// TwinCAT 3 PLC project Runtime
// ProgramVersion: 3.1.4026.14
// libraries:
//   Tc2_ControllerToolbox, * (Beckhoff Automation GmbH)
//   Tc2_ModbusSrv, * (Beckhoff Automation GmbH)
//   Tc2_Standard, * (Beckhoff Automation GmbH)
//   Tc2_System, * (Beckhoff Automation GmbH)
//   Tc2_Utilities, * (Beckhoff Automation GmbH)
//   Tc3_IotBase, * (Beckhoff Automation GmbH)
//   Tc3_Module, * (Beckhoff Automation GmbH)
// project tree:
//   DUTs/Algorithms/ stBESS.TcDUT, stCMD_SET.TcDUT, stCONV_UNION.TcDUT, stGRID_POS.TcDUT, stINVERTER.TcDUT, stMETER.TcDUT, stPF_POINT.TcDUT, stPOWER_PLANT.TcDUT, stPPC.TcDUT, stQV_POINT.TcDUT, stRECORD.TcDUT, stTIMESLOT.TcDUT
//   / FreqReg.TcTTO, PlcTask.TcTTO
//   GVLs/Algorithms/ GVL.TcGVL, GVL_Act_Pwr.TcGVL, GVL_Freq.TcGVL, GVL_Load_Following.TcGVL, GVL_Modules.TcGVL, GVL_React_Pwr.TcGVL, GVL_Voltage.TcGVL
//   POUs/ MAIN.TcPOU
//   POUs/Programs/Algorithms/Active power regulation/ Active_Power_Regulation.TcPOU, deltaActivePwr_Frequency_Regulation.TcPOU, FB_Frequency_Regulation.TcPOU, FB_Reach_SP_ActP.TcPOU
//   POUs/Programs/Algorithms/Automatic controls/ FF_BLOCK.TcPOU, Low_Pass_Filter.TcPOU, FB_PI_Setpoint.TcPOU
//   POUs/Programs/Algorithms/Cosmo Eco/ Calculate_Opt_SOC_Based_On_Conditions.TcPOU, Calculate_Opt_SOC_No_Decrease.TcPOU, Calculate_Set_Point_Normal_Conditions.TcPOU, No_Decrease.TcPOU, No_Increase.TcPOU, No_Limit.TcPOU, Pre_Lim.TcPOU, Static.TcPOU
//   POUs/Programs/Algorithms/Load Following/ FB_Load_Following.TcPOU
//   POUs/Programs/Algorithms/ FB_Load_From_DB.TcPOU, Main_Algorithm.TcPOU, FB_Module_Executor.TcPOU, outputQV_regulation.TcPOU, power_at_nominal_freq.TcPOU, Primary_Regulations.TcPOU, reactp_sp_from_pf.TcPOU, setpoint_acquired.TcPOU, sp_input_reducer.TcPOU
//   POUs/Programs/Algorithms/Meter/ Update_Virtual_Meter.TcPOU
//   POUs/Programs/Algorithms/Reactive power regulation/ deltaReactivePwr_Voltage_Regulation.TcPOU, FB_Hysteresis.TcPOU, FB_Map_QV.TcPOU, FB_Reach_SP_ReactP.TcPOU, FB_ReactivePwr_Voltage_Ctrl.TcPOU, Reactive_Power_Regulation.TcPOU
//   POUs/Programs/Engine/Inverter Comm/ Apply_Setpoint.TcPOU, FB_Check_Inverter_Health.TcPOU, FB_Command_Dispatcher.TcPOU, FB_Comm_Setup.TcPOU
//   POUs/Programs/Engine/ MQTT_TSO_Comm.TcPOU, FB_Read_Meter.TcPOU, FB_Setup_Meter_Comm.TcPOU

CONFIGURATION Runtime
    RESOURCE PLC ON TwinCAT3
        TASK FreqReg(INTERVAL := T#100000us, PRIORITY := 1);
        TASK PlcTask(INTERVAL := T#10ms, PRIORITY := 20);
        PROGRAM Primary_Regulations WITH FreqReg : Primary_Regulations;
        PROGRAM MAIN WITH PlcTask : MAIN;
    END_RESOURCE
END_CONFIGURATION

// ---- DUTs/Algorithms/stBESS.TcDUT
TYPE stBESS :
STRUCT
	
	soc: REAL; // [0, 1]
	capacity: REAL;
	available_power: REAL;
	
	max_tolerable_soc: REAL;
	min_tolerable_soc: REAL;
	
	soc_to_remove_sp: REAL;
	
	max_opt_soc: REAL;
	min_opt_soc: REAL;
	
	min_soc: REAL;
	efficiency: REAL;
	
	min_working_soc: REAL;
	
END_STRUCT
END_TYPE

// ---- DUTs/Algorithms/stCMD_SET.TcDUT
TYPE stCMD_SET :
STRUCT
	command_for_battery: REAL;
	plant_sp: REAL;
END_STRUCT
END_TYPE

// ---- DUTs/Algorithms/stCONV_UNION.TcDUT
TYPE stCONV_UNION :
UNION
	prod_real: REAL;
	prod_w: ARRAY[1..2] of WORD;
END_UNION
END_TYPE

// ---- DUTs/Algorithms/stGRID_POS.TcDUT
{attribute 'qualified_only'}
{attribute 'strict'}
TYPE stGRID_POS :
(
	poi := 0,
	pu := 1
);
END_TYPE

// ---- DUTs/Algorithms/stINVERTER.TcDUT
TYPE stINVERTER :
STRUCT
	/// INVERTER STATUS
	health: UINT;	// 1 = health, 0 = fault
	
	/// ACTIVE POWER ///
	current_sp: REAL;
	target_prod: REAL; 
	active_pwr_nominal_pwr: REAL;
	sp_mem: REAL;
	sp_mem_q: REAL;
	
	/// REACTIVE POWER /// 
	current_sp_q: REAL;
	reactive_pwr_nominal_pwr: REAL;
	
	/// MODBUS COMM
	tcp_port: UINT;
	unit_id: BYTE;
	server_ip_addr: STRING(255);
	n_quantity_act_pwr: WORD;
	mb_addr_act_pwr: WORD;
	n_quantity_react_pwr: WORD;
	mb_addr_react_pwr: WORD;
	mb_h_addr: WORD;
	health_quantity: WORD;
	
	read_done: BOOL := FALSE;
	read_state: UINT := 0;
	
	write_done: BOOL := TRUE;
	write_state: UINT := 0;
	
	wBusy_actp: BOOL;
	wBusy_reactp: BOOL;
	
	comm_state: UINT;
	
END_STRUCT
END_TYPE

// ---- DUTs/Algorithms/stMETER.TcDUT
TYPE stMETER :
STRUCT
	
	/// MODBUS ///
	tcp_port: UINT := 9501;
	unit_id: BYTE;
	server_ip_addr: STRING(255);
	
	/// ACTIVE POWER ///
	frequency: REAL;
	active_power_prod: REAL;
	active_power_sp: REAL;
	nQuantity_Act_Pwr: WORD;
	nMBAddr_Act_Pwr: WORD;
	
	/// REACTIVE POWER ///
	reactive_power_prod: REAL;
	reactive_power_sp: REAL;
	measured_voltage: REAL;
	nQuantity_React_Pwr: WORD;
	nMBAddr_React_Pwr: WORD;
	
	pos: stGRID_POS;	// questa variabile specifica dove è installato l'inverter e consente di distinguere meter di griglia (poi) da meter d'impianto (pu)
	
END_STRUCT
END_TYPE

// ---- DUTs/Algorithms/stPF_POINT.TcDUT
TYPE stPF_POINT :
STRUCT
	active_power: REAL;
	frequency: REAL;
END_STRUCT
END_TYPE

// ---- DUTs/Algorithms/stPOWER_PLANT.TcDUT
TYPE stPOWER_PLANT :
STRUCT
	// TO DO: in futuro, spostare tutte le variabili riguardanti l'impianto qui dentro
	safety_margin: REAL;
	max_power_increase: REAL; 
	ramp_limit: REAL; //[kW/min]
	sample_time: REAL;
	current_time: REAL;
	
	max_kw_change_3s: REAL;		// TO DO: questa variabile è rappresenta un'ulteriore limitazione che può essere presente in alcuni casi
	
	nominal_power: REAL := 1E4;
	
	avg_prod: REAL; 	// floating average level of production
	avg_prod_diff: REAL;
	
	avg_prod_3h: REAL; 	// average level of production over 3 hours. This variable is specific for the CosmoEco project 
	std_deviation_prod: REAL;
	
END_STRUCT
END_TYPE

// ---- DUTs/Algorithms/stPPC.TcDUT
TYPE stPPC :
STRUCT
	
	START: BOOL := TRUE;	
	MANUAL_MODE: BOOL;  /// FIELD OPERATOR ///
	AUTO_MODE: BOOL;	/// CONTROL ROOM ///
	REMOTE_MODE: BOOL := TRUE;	/// TSO via MQTT///
	
	actp_freq_reg_enabled: BOOL := FALSE;
	active_power_ctrl_enabled: BOOL := TRUE;
	reactive_power_ctrl_enabled: BOOL := TRUE;
	qv_ctrl_enabled: BOOL := TRUE;
	power_factor_ctrl_enabled: BOOL := FALSE;
	load_following_enabled: BOOL := FALSE;
	
	timeslot: stTIMESLOT;
	
END_STRUCT
END_TYPE

// ---- DUTs/Algorithms/stQV_POINT.TcDUT
TYPE stQV_POINT :
STRUCT
	voltage_ratio: REAL;
	q_pnd_ratio: REAL;
END_STRUCT
END_TYPE

// ---- DUTs/Algorithms/stRECORD.TcDUT
TYPE stRECORD :
STRUCT
	sp_value: REAL;
END_STRUCT
END_TYPE

// ---- DUTs/Algorithms/stTIMESLOT.TcDUT
TYPE stTIMESLOT :
STRUCT
	name: STRING(255);
	next: STRING(255);
	start: REAL;
	end: REAL;
END_STRUCT
END_TYPE

// ---- GVLs/Algorithms/GVL.TcGVL
//// POWER PLANT PARAMETERS ////

VAR_GLOBAL CONSTANT
	n_slave: UINT := 4;
	n_meter: UINT := 2;
	initial_tcp_port: UINT := 9501;
	server_addr: STRING := '127.0.0.1';
	
	n_meter_poi: UINT := 1;
	n_meter_pu: UINT := 1; 
	
	/// MQTT ///
	max_message_info: UINT := 5; 
END_VAR

VAR_GLOBAL
	/// INVERTER PARAMETERS ///
	inv: ARRAY[1..n_slave] OF stINVERTER;
	VIRTUAL_METER: stMETER;	/// questo è un meter di impianto
	meter_arr: ARRAY[1..n_meter] OF stMETER;
	healthy_inv: UINT := n_slave;
	
	/// POWER PLANT PARAMETERS - ACTIVE POWER - ///
	overall_current_prod: REAL := 0;
	power_plant_max_sp: REAL := 1;
	power_plant_max_sp_increase: REAL := 0.25;
	
	plant_sp_alpha: REAL := 0.4;
	
	/// POWER PLANT PARAMETERS - REACTIVE POWER - ///
	ReactP_PwrSp: REAL;
	power_plant_max_sp_q: REAL := 1;
	power_plant_max_sp_increase_q: REAL := 0.25;
	sp_tolerance_q : REAL := 0.002;	
	
	/// WISNAM PPC ///
	WISNAM_PPC: stPPC;
	
	/// MQTT /// 
	
	/// COSMO ECO ///
	windfarm_time: REAL;
	
	
	power_plant: stPOWER_PLANT;
	VIRTUAL_POI_METER: stMETER; /// meter di griglia
	battery: stBESS;
	
END_VAR

// ---- GVLs/Algorithms/GVL_Act_Pwr.TcGVL
VAR_GLOBAL
	
	/// ACTIVE POWER REGULATION ///
	target_prod: REAL;
	setpoint: REAL;
	total_sp: REAL;
	setpoint_mem: REAL;
	expected_pod_prod: REAL;
	setpoint_to_send: REAL;
	error_pi: REAL;
	pi_correction: REAL;
	setpoint_to_send_feed_forward: REAL;
	filtered_setpoint: REAL;
	low_pass_filter_mem: REAL;
	ff_pi_control_enable: BOOL := FALSE;
	active_p_ctrl_case: UINT := 1;
	setpoint_alpha: REAL := 0.1;
	sp_tolerance: REAL := 0.002;
	
	setpoint_manual: REAL;
	setpoint_auto: REAL;
	setpoint_tso: REAL;
	
	time_limit_sp_application: TIME := T#20S;
	ramp_rate_ctrl: BOOL := TRUE;
	ramp_rate_follow_inv: BOOL := TRUE;
	
	pi_ctrl_max_output: REAL := 1;
	pi_ctrl_min_output: REAL := -1;
	
	freq_reg_sp: REAL;	//setpoint derivante dalla regolazione in frequenza
END_VAR

// ---- GVLs/Algorithms/GVL_Freq.TcGVL
VAR_GLOBAL CONSTANT
	n_points: UINT;
END_VAR

VAR_GLOBAL
	/// FREQUENCY REGULATION ///
	output_pf_regulation: REAL;
	output_pf_regulation_scaled: REAL;
	frequency_smoothed: REAL;
	frequency_smoothed_mem: REAL;
	p_nd: REAL;
	
	K_FSMU: REAL := 0.5;
	K_FSMO: REAL := 0.5;
	frequency_reference: REAL := 50;
	
	enhanced_points: ARRAY [1..n_points, 1..3] OF REAL;
	out_limiter_max: REAL := 1.0;
	out_limiter_min: REAL := -1.0;
	
	under_f_db_threshold: REAL := 49.980;
	over_f_db_threshold: REAL := 50.020;
	
	over_f_medium_threshold: REAL := 50.20;
	under_f_medium_threshold: REAL := 49.8;
	
	max_value_over_f: REAL := 51.5;
	min_value_under_f: REAL := 49.5;
	
	S_under_mid_val: REAL :=  2.5;
	S_over_mid_val: REAL := 2.5;
	S_under_ext_val: REAL := 2.5;
	S_over_ext_val: REAL := 2.5;
	
	frequency_regulation_priority: BOOL;
	sp_nominal_freq: REAL;
	max_delta_sp: REAL := 0.25;
	prod_nominal_freq: REAL;
	
	n_pf_soil: UINT; // numero di soglie di power factor
	pf_conf: ARRAY[1..3] OF ARRAY[1..2]  OF REAL := [[0.5, 0.98], [0.7, 0.95], [1, 0.93]];
	
END_VAR

// ---- GVLs/Algorithms/GVL_Load_Following.TcGVL
VAR_GLOBAL
	
	p_sp: REAL;
	
	delta: REAL := 1E-2;
	delta_fast: REAL := 1.5E-2;
	delta_slow: REAL := 0.8E-2;
	
	p_sp_max: REAL;
	p_sp_min: REAL;
	
	power_grid_min: REAL := 5000;
	power_grid_max: REAL := 8000;
	
	max_error_perc: REAL := 40;
	
END_VAR

// ---- GVLs/Algorithms/GVL_Modules.TcGVL
VAR_GLOBAL CONSTANT
	n_modules: UINT := 7;
END_VAR
VAR_GLOBAL
	read_meter: STRING(255) := 'read_meter';
	check_inverter_health: STRING(255) := 'check_inverter_health';
	active_power_ctrl: STRING(255) := 'active_power_ctrl'; 
	reactive_power_ctrl: STRING(255) := 'reactive_power_ctrl';
	command_dispatcher: STRING(255) := 'command_dispatcher';
	acquire_setpoint_mqtt: STRING(255) := 'acquire_setpoint_mqtt';
	load_following: STRING(255) := 'load_following';
END_VAR

// ---- GVLs/Algorithms/GVL_React_Pwr.TcGVL
VAR_GLOBAL CONSTANT
	n_points: UINT;
END_VAR

VAR_GLOBAL
	/// REACTIVE POWER REGULATION /// 
	setpoint: REAL;
	total_sp: REAL;
	target_prod: REAL;
	expected_pod_prod_q: REAL;
	setpoint_mem: REAL;
	reactive_pwr_ctrl_case: UINT := 1;
	setpoint_ff: REAL;
	filtered_setpoint: REAL;
	low_pass_filter_mem_q: REAL;
	update_pi_sp_q: FB_PI_Setpoint;
	pi_correction_q: REAL;
	ff_pi_q_control_enable: BOOL;
	setpoint_to_send: REAL;
	setpoint_alpha: REAL := 0.2;
	sp_tolerance_q: REAL := 0.002;
	
	setpoint_manual: REAL;
	setpoint_auto: REAL;
	setpoint_tso: REAL;
	p_nd: REAL;
	
	max_q_pf_regulation: REAL;
	
	power_factor_target: REAL := 1.0;
	//enhanced_points: ARRAY [1..n_points, 1..2] OF REAL := [[-0.35, 0], [0, 1.1], [0.35, 1.05], [0, 0.9]];
	voltage_hyst_enable: BOOL;
END_VAR

// ---- GVLs/Algorithms/GVL_Voltage.TcGVL
VAR_GLOBAL
	reference_value: REAL := 1000;
	measured_value: REAL;
	error: REAL;
	norm_error: REAL;
	max_norm_correction: REAL := 0.35;
	min_norm_correction: REAL := -0.35;
	output_qv_regulation: REAL;
	last_output_qv_regulation: REAL;
	output_pi: REAL;
	pi_ctrl_max_output: REAL := 1;
	pi_ctrl_min_output: REAL := -1;
	hyst_clearance: REAL := 0.01;	// isteresi TO DO: controlla questo parametro 
	v_norm: REAL;
	
	// QV map vertices [-0.1, 0.33], [-0.01, 0.0], [0.01, 0.0], [0.1, -0.33]
END_VAR

// ---- POUs/Programs/Algorithms/Primary_Regulations.TcPOU
PROGRAM Primary_Regulations
VAR
	f_error: REAL;
	power_percentage_delta: REAL;
	overshoot_freq_error: REAL;
	delta_p: REAL;
	available_power: REAL;
	reach_sp: FB_Reach_SP_ActP;
	command_dispatcher: FB_Command_Dispatcher;
	i: UINT;
	current_pf: REAL;
	phi: REAL;
	
	
END_VAR

IF GVL.WISNAM_PPC.power_factor_ctrl_enabled THEN
	
	reactp_sp_from_pf();	

END_IF

IF GVL.WISNAM_PPC.actp_freq_reg_enabled THEN

	power_at_nominal_freq();
	IF GVL_Freq.frequency_regulation_priority THEN
		
		GVL_Act_Pwr.setpoint_to_send := GVL_Act_Pwr.freq_reg_sp;
		
	END_IF
		
END_IF


IF GVL.WISNAM_PPC.qv_ctrl_enabled THEN
	
	GVL_React_Pwr.setpoint_to_send := outputQV_regulation();

END_IF


IF GVL.WISNAM_PPC.actp_freq_reg_enabled AND GVL.WISNAM_PPC.power_factor_ctrl_enabled THEN
	
	GVL_React_Pwr.total_sp := MIN(GVL_React_PWr.max_q_pf_regulation, GVL_React_Pwr.total_sp);

END_IF


command_dispatcher();

END_PROGRAM

// ---- POUs/Programs/Algorithms/Active power regulation/FB_Reach_SP_ActP.TcPOU
FUNCTION_BLOCK FB_Reach_SP_ActP
VAR_INPUT
	sp_target_actp: REAL;
END_VAR
VAR_OUTPUT
END_VAR
VAR
	update_pi_sp: FB_PI_Setpoint;
	low_pass_filter_mem: REAL;
	setpoint_to_send_ff: REAL;
	filtered_sp: REAL;
	pi_correction: REAL;
END_VAR

IF ABS(GVL.VIRTUAL_METER.active_power_sp - sp_target_actp) > GVL_Act_Pwr.sp_tolerance THEN
	
	IF GVL_Act_Pwr.ff_pi_control_enable THEN
		
		/// 10. FEED FORWARD REGULATOR ///
		setpoint_to_send_ff := FF_BLOCK(input_value := sp_target_actp, k_ff := 0.025);

		/// 9. LOW PASS FILTER + 12. FEEDBACK ///
		filtered_sp := Low_Pass_Filter(plant_target := sp_target_actp, filter_output_mem := low_pass_filter_mem, alpha := GVL_Act_Pwr.setpoint_alpha);
		sp_target_actp := filtered_sp;

		update_pi_sp(sp_value := filtered_sp, feedback_sp := GVL.VIRTUAL_METER.active_power_sp, pi_output => pi_correction);
	
		/// 13. TOTAL PLANT COMMAND ///
		GVL_Act_Pwr.setpoint_to_send := setpoint_to_send_ff + pi_correction;
		GVL_Act_Pwr.expected_pod_prod := GVL_Act_Pwr.setpoint_to_send*GVL.power_plant.nominal_power;
		
	ELSE
		CASE GVL_Act_Pwr.active_p_ctrl_case OF
			1: 
				// update setpoint
				IF GVL_Act_Pwr.ramp_rate_follow_inv THEN	// TO DO: approfondire il discorso dell'irraggiamento
					GVL_Act_Pwr.setpoint_to_send := GVL_Act_Pwr.setpoint_alpha * sp_target_actp + (1 - GVL_Act_Pwr.setpoint_alpha)*GVL.VIRTUAL_METER.active_power_sp;
					GVL_Act_Pwr.expected_pod_prod := GVL_Act_Pwr.setpoint_to_send*GVL.power_plant.nominal_power;
					GVL_Act_Pwr.active_p_ctrl_case := 2;
					GVL_Act_Pwr.setpoint_mem := GVL_Act_Pwr.setpoint;
				END_IF
				
			2:
				// wait until the plant is close to current setpoint
				//timer_sp(IN := (ABS(GVL_Act_Pwr.setpoint_to_send - GVL.VIRTUAL_METER.active_power_sp) > 0.025), PT := GVL_Act_Pwr.time_limit_sp_application, Q =>);
				IF ABS(GVL_Act_Pwr.setpoint_to_send - GVL.VIRTUAL_METER.active_power_sp) < 0.1 THEN
					
					GVL_Act_Pwr.active_p_ctrl_case := 1;
					//timer_sp(IN := FALSE);
					
				ELSE
					
//						IF timer_sp.Q THEN
//							timer_sp(IN := FALSE);
//							GVL_Act_Pwr.setpoint := GVL.VIRTUAL_METER.active_power_sp;
//							GVL_Act_Pwr.setpoint_to_send := GVL.VIRTUAL_METER.active_power_sp;
//							GVL_Act_Pwr.ramp_rate_ctrl := FALSE;
//							GVL_Act_Pwr.ramp_rate_follow_inv := FALSE;
//							GVL_Act_Pwr.setpoint_mem := GVL_Act_Pwr.setpoint_to_send;
//						END_IF
				END_IF
	
			3:
				// fault management
		END_CASE
		
	END_IF

	IF GVL_Act_Pwr.expected_pod_prod > GVL.power_plant.nominal_power THEN
		GVL_Act_Pwr.setpoint_to_send := 1;
		GVL_Act_Pwr.expected_pod_prod := GVL.power_plant.nominal_power;
	END_IF 
	
END_IF

END_FUNCTION_BLOCK

// ---- POUs/Programs/Algorithms/Automatic controls/FB_PI_Setpoint.TcPOU
FUNCTION_BLOCK FB_PI_Setpoint
VAR_IN_OUT
	feedback_sp: REAL;
END_VAR
VAR_INPUT
	sp_value: REAL;
END_VAR
VAR_OUTPUT
	pi_output: REAL;
END_VAR
VAR
	fbCTRL_PI: FB_CTRL_PI;
	stCTRL_PI_PARAMS: ST_CTRL_PI_PARAMS;
	eMode: E_CTRL_MODE;
	bInit: BOOL := TRUE;
	fbTON: TON;
	f_out: REAL;
	activatePI: BOOL := TRUE;
END_VAR

IF bInit THEN
	(* init parameter struct *)
	stCTRL_PI_PARAMS.tCtrlCycleTime		:= T#50MS;		// TO DO: parametrizza questi valori
	stCTRL_PI_PARAMS.tTaskCycleTime		:= T#10MS;
	stCTRL_PI_PARAMS.tTn				:= T#2000MS;		(* integral gain Tn				*)
	stCTRL_PI_PARAMS.fKp				:= 0.04;			(* proportional gain Kp				*)
	stCTRL_PI_PARAMS.fOutMaxLimit		:=  GVL_Act_Pwr.pi_ctrl_max_output;  		(* maximum output limit				*)
	stCTRL_PI_PARAMS.fOutMinLimit		:=  GVL_Act_Pwr.pi_ctrl_min_output;			(* minimum output limit				*)

	(* set the mode to ACTIVE --> normal operation *)
	eMode := eCTRL_MODE_ACTIVE;

	(* reset the init flag *)
	bInit := FALSE;
END_IF

IF activatePI THEN
	fbCTRL_PI(
		fSetpointValue:= sp_value, 
		fActualValue:= feedback_sp, 
		fManSyncValue:= , 
		bSync:= , 
		eMode:= eMode, 
		bHold:= , 
		fOut=> pi_output, 
		bARWactive=> , 
		eState=> , 
		eErrorId=> , 
		bError=> , 
		stParams:= stCTRL_PI_PARAMS
	);
END_IF

END_FUNCTION_BLOCK

// ---- POUs/Programs/Algorithms/Automatic controls/FF_BLOCK.TcPOU
FUNCTION FF_BLOCK : REAL
VAR_INPUT
	input_value: REAL;
	k_ff: REAL;
END_VAR
VAR
END_VAR

FF_BLOCK := input_value * (1 + k_ff);

END_FUNCTION

// ---- POUs/Programs/Algorithms/Automatic controls/Low_Pass_Filter.TcPOU
FUNCTION Low_Pass_Filter : REAL
VAR_IN_OUT
	plant_target: REAL;
	filter_output_mem: REAL;
	alpha: REAL;
END_VAR

Low_Pass_Filter := alpha*plant_target + (1-alpha)*filter_output_mem;

END_FUNCTION

// ---- POUs/Programs/Engine/Inverter Comm/FB_Command_Dispatcher.TcPOU
FUNCTION_BLOCK FB_Command_Dispatcher
VAR_INPUT
END_VAR
VAR_OUTPUT
END_VAR
VAR
	check_inverter_health: FB_MBReadRegs;
	aux_union: stCONV_UNION;
	aux_union_q: stCONV_UNION;
	fb_write_holding_actp: FB_MBWriteRegs;
	fb_write_holding_reactp: FB_MBWriteRegs;
	comm_state: UINT;
	index: UINT;
END_VAR

CASE comm_state OF

	0:
		index := 1;
		comm_state := 1;
		GVL.healthy_inv := 0;

	1:
		check_inverter_health(
			sIPAddr:= GVL.server_addr, 
			nTCPPort:= GVL.inv[index].tcp_port, 
			nUnitID:= GVL.inv[index].unit_id, 
			nQuantity:= GVL.inv[index].health_quantity, 
			nMBAddr:= GVL.inv[index].mb_h_addr, 
			cbLength:= SIZEOF(GVL.inv[index].health), 
			pDestAddr:= ADR(GVL.inv[index].health), 
			bExecute:= TRUE, 
			tTimeout:= T#2S, 
			bBusy=> , 
			bError=> , 
			nErrId=> , 
			cbRead=> 
		);
		comm_state := 2;

	2:
		check_inverter_health(bExecute := FALSE);
		IF NOT check_inverter_health.bBusy THEN
			IF check_inverter_health.bError THEN
				GVL.inv[index].health := 0;
			END_IF
			comm_state := 3;
		END_IF

	3:
		GVL.healthy_inv := GVL.healthy_inv + GVL.inv[index].health;
		index := index + 1;
		
		IF index > GVL.n_slave THEN
			index := 1;
			comm_state := 4;
		ELSE
			comm_state := 1;
		END_IF

	4:
		IF (GVL.WISNAM_PPC.active_power_ctrl_enabled) AND GVL.healthy_inv <> 0 AND GVL.inv[index].health = 1 THEN
			GVL.inv[index].current_sp := ((GVL_Act_Pwr.setpoint_to_send * GVL.power_plant.nominal_power)/UINT_TO_REAL(GVL.healthy_inv))/GVL.inv[index].active_pwr_nominal_pwr;
			GVL.inv[index].current_sp := MIN(1, MAX(GVL.inv[index].current_sp,0));
			IF GVL.inv[index].sp_mem <> GVL.inv[index].current_sp THEN
				
				aux_union.prod_real := GVL.inv[index].current_sp;
				fb_write_holding_actp(
					sIPAddr:= GVL.server_addr, 
					nTCPPort:= GVL.inv[index].tcp_port, 
					nUnitID:= GVL.inv[index].unit_id, 
					nQuantity:= GVL.inv[index].n_quantity_act_pwr, 
					nMBAddr:= GVL.inv[index].mb_addr_act_pwr, 
					cbLength:= SIZEOF(DWORD), 
					pSrcAddr:= ADR(aux_union.prod_w), 
					bExecute:= TRUE, 
					tTimeout:= T#3S, 
					bBusy=> , 
					bError=> , 
					nErrId=>
				);
				GVL.inv[index].sp_mem := GVL.inv[index].current_sp;
				
			END_IF
			
		END_IF
		
		IF (GVL.WISNAM_PPC.reactive_power_ctrl_enabled) AND GVL.healthy_inv <> 0 AND GVL.inv[index].health = 1 THEN
			GVL.inv[index].current_sp_q := ((GVL_React_Pwr.setpoint_to_send * GVL.power_plant.nominal_power) / UINT_TO_REAL(GVL.healthy_inv))/GVL.inv[index].active_pwr_nominal_pwr;
			GVL.inv[index].current_sp_q := MIN(1, MAX(GVL.inv[index].current_sp_q,0));
			IF GVL.inv[index].sp_mem_q <> GVL.inv[index].current_sp_q THEN
				
				aux_union_q.prod_real := GVL.inv[index].current_sp_q;
				fb_write_holding_reactp(
					sIPAddr:= GVL.server_addr, 
					nTCPPort:= GVL.inv[index].tcp_port, 
					nUnitID:= GVL.inv[index].unit_id, 
					nQuantity:= GVL.inv[index].n_quantity_react_pwr, 
					nMBAddr:= GVL.inv[index].mb_addr_react_pwr, 
					cbLength:= SIZEOF(DWORD), 
					pSrcAddr:= ADR(aux_union_q.prod_w), 
					bExecute:= TRUE, 
					tTimeout:= T#3S, 
					bBusy=> , 
					bError=> , 
					nErrId=>
				);
				GVL.inv[index].sp_mem_q := GVL.inv[index].current_sp_q;
				
			END_IF
			
		END_IF
		// TO DO: valutare se realizzare due stati separati per le due scritture
		comm_state := 5;

	5:
		fb_write_holding_actp(bExecute := FALSE);
		fb_write_holding_reactp(bExecute := FALSE);
		IF NOT fb_write_holding_actp.bBusy AND NOT fb_write_holding_reactp.bBusy THEN
			comm_state := 6; 
		END_IF

	6:
		index := index + 1;
		IF index > GVL.n_slave THEN
			comm_state := 0;
		ELSE
			comm_state := 4;
		END_IF

END_CASE

END_FUNCTION_BLOCK

// ---- POUs/Programs/Algorithms/reactp_sp_from_pf.TcPOU
FUNCTION reactp_sp_from_pf : real
VAR_INPUT
END_VAR
VAR
	current_pf: REAL;
	i: UINT;
	phi: REAL;
END_VAR

current_pf := -1;

IF GVL.WISNAM_PPC.power_factor_ctrl_enabled THEN
	
	FOR i := 1 TO GVL_Freq.n_pf_soil DO
	
		IF (GVL.VIRTUAL_METER.active_power_sp < GVL_Freq.pf_conf[i][1]) AND current_pf = -1 THEN
			
			current_pf := GVL_Freq.pf_conf[i][2];
			
		END_IF	
	
	END_FOR 	
	
	phi := ACOS(current_pf);
	GVL_React_Pwr.max_q_pf_regulation := GVL.VIRTUAL_METER.active_power_sp * TAN(phi);
		
END_IF

END_FUNCTION

// ---- POUs/Programs/Algorithms/power_at_nominal_freq.TcPOU
FUNCTION power_at_nominal_freq : real
VAR_INPUT
END_VAR
VAR
	available_power: REAL;
	f_error: REAL;
	power_percentage_delta: REAL;
	overshoot_freq_error: REAL;
	delta_p: REAL;
END_VAR

available_power := GVL_Freq.p_nd * GVL.power_plant.nominal_power;
GVL_Act_Pwr.freq_reg_sp := GVL.VIRTUAL_METER.active_power_prod;

/// dead-band ////////////////////////////////////////////
IF GVL_Freq.under_f_db_threshold <= GVL.VIRTUAL_METER.frequency AND GVL.VIRTUAL_METER.frequency <= GVL_Freq.over_f_db_threshold THEN
	GVL_Freq.frequency_regulation_priority := FALSE;	
	GVL_Act_Pwr.freq_reg_sp := GVL.VIRTUAL_METER.active_power_sp;
	RETURN;
END_IF
/////////////////////////////////////////////////////////

/// critical scenarios /////////////////////////////////
IF GVL.VIRTUAL_METER.frequency > GVL_Freq.max_value_over_f THEN
	GVL_Act_Pwr.freq_reg_sp := 0;
	GVL_Freq.frequency_regulation_priority := TRUE;
	RETURN;
END_IF


IF GVL.VIRTUAL_METER.frequency < GVL_Freq.min_value_under_f THEN
	GVL_Act_Pwr.freq_reg_sp := 1;
	GVL_Freq.frequency_regulation_priority := TRUE;
	RETURN;
END_IF
/////////////////////////////////////////////////////////


/// FSM-O ///////////////////////////////////////////////
IF GVL_Freq.over_f_db_threshold < GVL.VIRTUAL_METER.frequency AND GVL.VIRTUAL_METER.frequency <= GVL_Freq.over_f_medium_threshold THEN
	GVL_Freq.frequency_regulation_priority := TRUE;
	f_error := ABS(GVL.VIRTUAL_METER.frequency - GVL_Freq.frequency_reference);
	power_percentage_delta := f_error*GVL_Freq.S_over_mid_val;
END_IF
/////////////////////////////////////////////////////////


/// FSM-U ///////////////////////////////////////////////
IF GVL_Freq.under_f_db_threshold > GVL.VIRTUAL_METER.frequency AND GVL.VIRTUAL_METER.frequency >= GVL_Freq.under_f_medium_threshold THEN
	GVL_Freq.frequency_regulation_priority := TRUE;
	f_error := ABS(GVL.VIRTUAL_METER.frequency - GVL_Freq.frequency_reference);
	power_percentage_delta := f_error*GVL_Freq.S_under_mid_val;
END_IF
/////////////////////////////////////////////////////////


/// LFSM-O //////////////////////////////////////////////
IF GVL_Freq.over_f_medium_threshold < GVL.VIRTUAL_METER.frequency THEN
	GVL_Freq.frequency_regulation_priority := TRUE;
	f_error := ABS(GVL.VIRTUAL_METER.frequency - GVL_Freq.frequency_reference);
	overshoot_freq_error := ABS(GVL_Freq.over_f_medium_threshold - GVL_Freq.over_f_db_threshold)/20; // TO DO: parametrizzare
	power_percentage_delta := (f_error + overshoot_freq_error)*GVL_Freq.S_over_ext_val;
END_IF
/////////////////////////////////////////////////////////


/// LFSM-U //////////////////////////////////////////////
IF GVL_Freq.under_f_medium_threshold > GVL.VIRTUAL_METER.frequency THEN
	GVL_Freq.frequency_regulation_priority := TRUE;
	f_error := ABS(GVL.VIRTUAL_METER.frequency - GVL_Freq.frequency_reference);
	overshoot_freq_error := ABS(GVL_Freq.under_f_medium_threshold - GVL_Freq.under_f_db_threshold)/20; // TO DO: parametrizzare
	power_percentage_delta := (f_error + overshoot_freq_error)*GVL_Freq.S_over_ext_val;	
END_IF
/////////////////////////////////////////////////////////

IF (power_percentage_delta / 100) > GVL_Freq.max_delta_sp THEN
	
	power_percentage_delta := GVL_Freq.max_delta_sp * 100;
	
END_IF	

delta_p := (available_power/100) * power_percentage_delta;

IF GVL.VIRTUAL_METER.frequency > GVL_Freq.frequency_reference THEN
	GVL_Act_Pwr.freq_reg_sp := GVL.VIRTUAL_METER.active_power_prod - delta_p;
ELSE
	GVL_Act_Pwr.freq_reg_sp := GVL.VIRTUAL_METER.active_power_prod + delta_p;
END_IF


//reach_sp(sp_target_actp := GVL_Act_Pwr.freq_reg_sp);
GVL_Act_Pwr.freq_reg_sp := GVL_Act_Pwr.freq_reg_sp / GVL.power_plant.nominal_power;

END_FUNCTION

// ---- POUs/Programs/Algorithms/outputQV_regulation.TcPOU
FUNCTION outputQV_regulation : real
VAR_INPUT
END_VAR
VAR
	current_v: REAL;
	v_nom: REAL := 1000;
	deadband: REAL := 0.05;
	hyst: REAL := 0.02;
	statism: REAL := 3;	// [0, 100] %
	increment_threshold: REAL := 0.08;
	q_max_variation: REAL := 0.2;
	q_fixed_increment: REAL := 0.005;
	
	lower_db: REAL := v_nom - deadband * v_nom;
	upper_db: REAL := v_nom + deadband * v_nom;
	
	lower_hyst: REAL := v_nom * (1 - hyst);
	upper_hyst: REAL := v_nom * (1 + hyst);
	
	lower_inc_th: REAL := v_nom - increment_threshold;
	upper_inc_th: REAL := v_nom + increment_threshold;
	
	v_error: REAL;
	q_delta: REAL;
	
	norm_s: REAL;
END_VAR

current_v := GVL.VIRTUAL_METER.measured_voltage;

IF current_v < lower_db OR current_v > upper_db THEN
	
	GVL_React_Pwr.voltage_hyst_enable := TRUE;

END_IF


IF GVL_React_Pwr.voltage_hyst_enable THEN
	
	IF lower_hyst < current_v AND current_v < upper_hyst THEN
		
		GVL_React_Pwr.voltage_hyst_enable := FALSE;
		outputQV_regulation := GVL.VIRTUAL_METER.reactive_power_sp;
		RETURN;
	
	END_IF

	
	IF current_v < lower_hyst THEN
		
		IF current_v < lower_inc_th THEN
			
			v_error := ABS(v_nom - current_v);
			norm_s := statism / 100 ;
			q_delta := MIN(v_error * norm_s, q_max_variation);
			outputQV_regulation := GVL.VIRTUAL_METER.reactive_power_sp + q_delta;
			RETURN;
			
		ELSE
			
			outputQV_regulation := GVL.VIRTUAL_METER.reactive_power_sp + q_fixed_increment;
			RETURN;
			
		END_IF
	
	END_IF
	
	
	IF current_v > upper_hyst THEN
		
		IF current_v > upper_inc_th THEN
			
			v_error := ABS(v_nom - current_v);
			norm_s := statism / 100 ;
			q_delta := MIN(v_error * norm_s, q_max_variation);
			outputQV_regulation := GVL.VIRTUAL_METER.reactive_power_sp - q_delta;
			RETURN;
			
		ELSE
	
			outputQV_regulation := GVL.VIRTUAL_METER.reactive_power_sp - q_fixed_increment;
			RETURN;
	
		END_IF
	
	END_IF
	
END_IF

outputQV_regulation := GVL.VIRTUAL_METER.reactive_power_sp;

END_FUNCTION

// ---- POUs/MAIN.TcPOU
PROGRAM MAIN
VAR
END_VAR

Main_Algorithm();

END_PROGRAM

// ---- POUs/Programs/Algorithms/Main_Algorithm.TcPOU
PROGRAM Main_Algorithm
VAR
	module_executer: ARRAY[1..GVL_MODULES.n_modules] OF FB_Module_Executor;
	setup_inverter_comm: FB_Comm_Setup;
	setup_meter_comm: FB_Setup_Meter_Comm;
	i: UINT;
END_VAR

MAIN_1();
//MAIN_2();

METHOD MAIN_1 : BOOL
VAR_INPUT
END_VAR
VAR
	//load_from_db: LOAD_FROM_DB_FB;
END_VAR
IF GVL.WISNAM_PPC.START THEN			/// setup del simulatore ///
	setup_inverter_comm();
	setup_meter_comm();
	GVL.WISNAM_PPC.START := FALSE;
END_IF


module_executer[1](input := GVL_modules.read_meter);
module_executer[3](input := GVL_MODULES.acquire_setpoint_mqtt);
module_executer[4](input := GVL_modules.active_power_ctrl);
module_executer[5](input := GVL_modules.reactive_power_ctrl);
//IF NOT GVL_Freq.frequency_regulation_priority OR NOT GVL.WISNAM_PPC.actp_freq_reg_enabled THEN
//	module_executer[6](input := GVL_modules.command_dispatcher);
//END_IF
// load_from_db();
// test
END_METHOD

METHOD MAIN_2 : BOOL
VAR_INPUT
END_VAR
IF GVL.WISNAM_PPC.START THEN			/// setup del simulatore ///
	setup_inverter_comm();
	setup_meter_comm();
	GVL.WISNAM_PPC.START := FALSE;
END_IF


module_executer[1](input := GVL_modules.read_meter);
Update_Virtual_Meter();
module_executer[3](input := GVL_MODULES.acquire_setpoint_mqtt);
module_executer[4](input := GVL_modules.load_following);
module_executer[5](input := GVL_modules.reactive_power_ctrl);
module_executer[6](input := GVL_modules.command_dispatcher);
END_METHOD

METHOD MAIN_WIND_BESS : BOOL
VAR_INPUT
END_VAR
/// per tutte le funzioni "derivate" dal progetto originale Cosmo Eco, la potenza è espressa in termini assoluti e poi normalizzata qui ///
/// TO DO: valutare se mantenere questo approccio ///

/// Ciascuna delle funzioni richiamate restituisce variabili di tipo COMMAND SET (CMD_SET) 
/// TO DO: definire (lato progettazione) come devono essere ripartiti questi comandi e da quali moduli
/// Tutti questi moduli devono essere ridisegnati in fase di progettazione per l'interfacciamento con un sistema reale
END_METHOD

END_PROGRAM

// ---- POUs/Programs/Algorithms/FB_Module_Executor.TcPOU
FUNCTION_BLOCK FB_Module_Executor
VAR_INPUT
	input: STRING(255);
END_VAR
VAR_OUTPUT
END_VAR
VAR
	read_meter: ARRAY[1..GVL.n_meter] OF FB_Read_Meter;
	check_inverter_health: FB_Check_Inverter_Health;
	active_power_ctrl: Active_Power_Regulation;
	reactive_power_ctrl: Reactive_Power_Regulation;
	acquire_setpoint_mqtt: MQTT_TSO_Comm;
	command_dispatcher: FB_Command_Dispatcher;
	load_following: FB_Load_Following;
	i: UINT;
END_VAR

IF input = TO_STRING("read_meter") THEN
	FOR i := 1 TO GVL.n_meter DO
		read_meter[i](tcp_port := GVL.meter_arr[i].tcp_port, nUnitID := GVL.meter_arr[i].unit_id, 
						nQuantity_Act_Pwr := GVL.meter_arr[i].nQuantity_Act_Pwr, nMBAddr_Act_Pwr := GVL.meter_arr[i].nMBAddr_Act_Pwr, 
						nQuantity_React_Pwr := GVL.meter_arr[i].nQuantity_React_Pwr, nMBAddr_React_Pwr := GVL.meter_arr[i].nMBAddr_React_Pwr,		
						i := i);	
	END_FOR
	Update_Virtual_Meter();
END_IF


IF input = TO_STRING("check_inverter_health") THEN
	check_inverter_health();
END_IF


IF input = TO_STRING("acquire_setpoint_mqtt") THEN
	acquire_setpoint_mqtt();
END_IF


IF input = TO_STRING("active_power_ctrl") THEN
	active_power_ctrl();
END_IF


IF input = TO_STRING("reactive_power_ctrl") THEN
	reactive_power_ctrl();
END_IF


IF input = TO_STRING("command_dispatcher") THEN
	command_dispatcher();
END_IF


IF input = TO_STRING("load_following") THEN
	load_following();
END_IF

END_FUNCTION_BLOCK

// ---- POUs/Programs/Engine/FB_Read_Meter.TcPOU
FUNCTION_BLOCK FB_Read_Meter
VAR_INPUT
	tcp_port: UINT;
	nUnitID: BYTE;
	nQuantity_Act_Pwr: WORD;
	nMBAddr_Act_Pwr: WORD;
	nQuantity_React_Pwr: WORD;
	nMBAddr_React_Pwr: WORD;
	i: UINT;
END_VAR
VAR_OUTPUT
END_VAR
VAR
	/// MODBUS ///
	timer_read: TON;
	bBusy: BOOL;
	bError: BOOL;
	nErrID: UDINT;
	
	/// ACTIVE POWER ///
	aux_arr_active_pwr: ARRAY[1..4] OF WORD;
	convert_meter_active_pwr: stCONV_UNION;
	convert_meter_freq: stCONV_UNION;
	read_meter_prod_active_pwr: FB_MBReadRegs;
	
	/// REACTIVE POWER ///
	read_meter_prod_reactive_pwr: FB_MBReadRegs;
	aux_arr_reactive_pwr: ARRAY[1..4] OF WORD;
	convert_meter_reactive_pwr: stCONV_UNION;
	convert_meter_voltage: stCONV_UNION;
END_VAR

timer_read(IN := NOT timer_read.Q, PT := T#70MS, Q =>);
IF GVL.WISNAM_PPC.active_power_ctrl_enabled THEN
	
	read_meter_prod_active_pwr(
			sIPAddr:= GVL.server_addr, 
			nTCPPort:= tcp_port, 
			nUnitID:= nUnitID, 
			nQuantity:= nQuantity_Act_Pwr, 
			nMBAddr:= nMBAddr_Act_Pwr, 
			cbLength:= SIZEOF(aux_arr_active_pwr), 
			pDestAddr:= ADR(aux_arr_active_pwr), 
			bExecute:= timer_read.Q, 
			tTimeout:= T#3S, // TO DO parametrizza timeout lettura scrittera
			bBusy=> bBusy, 
			bError=> bError, 
			nErrId=> nErrID, 
			cbRead=> 
			);	
			
	convert_meter_active_pwr.prod_w[2] := aux_arr_active_pwr[1];
	convert_meter_active_pwr.prod_w[1] := aux_arr_active_pwr[2];
	GVL.meter_arr[i].active_power_prod := convert_meter_active_pwr.prod_real;
	GVL.meter_arr[i].active_power_sp := GVL.meter_arr[1].active_power_prod/GVL.power_plant.nominal_power;
	
	convert_meter_freq.prod_w[2] := aux_arr_active_pwr[3];
	convert_meter_freq.prod_w[1] := aux_arr_active_pwr[4];
	GVL.meter_arr[i].frequency := convert_meter_freq.prod_real;
	
END_IF

// TO DO: in generale, separa le letture di potenza attiva / frequenza e potenza reattiva / tensione

IF GVL.WISNAM_PPC.reactive_power_ctrl_enabled THEN
	
	read_meter_prod_reactive_pwr(
			sIPAddr:= GVL.server_addr, 
			nTCPPort:= tcp_port, 
			nUnitID:= nUnitID, 
			nQuantity:= nQuantity_React_Pwr, 
			nMBAddr:= nMBAddr_React_Pwr, 
			cbLength:= SIZEOF(aux_arr_reactive_pwr), 
			pDestAddr:= ADR(aux_arr_reactive_pwr), 
			bExecute:= timer_read.Q, 
			tTimeout:= T#3S, 
			bBusy=> bBusy, 
			bError=> bError, 
			nErrId=> nErrID, 
			cbRead=> 
			);	
	
	convert_meter_reactive_pwr.prod_w[2] := aux_arr_reactive_pwr[1];
	convert_meter_reactive_pwr.prod_w[1] := aux_arr_reactive_pwr[2];
	GVL.meter_arr[i].reactive_power_prod := convert_meter_reactive_pwr.prod_real;
	GVL.meter_arr[i].reactive_power_sp := GVL.meter_arr[1].reactive_power_prod/GVL.power_plant.nominal_power;
	
	convert_meter_voltage.prod_w[2] := aux_arr_reactive_pwr[3];
	convert_meter_voltage.prod_w[1] := aux_arr_reactive_pwr[4];
	GVL.meter_arr[i].measured_voltage := convert_meter_voltage.prod_real;
	
END_IF

END_FUNCTION_BLOCK

// ---- POUs/Programs/Engine/Inverter Comm/FB_Check_Inverter_Health.TcPOU
FUNCTION_BLOCK FB_Check_Inverter_Health
VAR_INPUT
END_VAR
VAR_OUTPUT
END_VAR
VAR
	i: UINT;
	timer_heart_beat: TON;
	check_inverter_health: ARRAY[1..GVL.n_slave] OF FB_MBReadRegs;
	regulating_timer: TON;
	new_check:  BOOL;
	all_done: BOOL;
END_VAR

IF NOT new_check THEN
    regulating_timer(IN := TRUE, PT := T#10S);
    IF regulating_timer.Q THEN
         new_check := TRUE;
         regulating_timer(IN := FALSE, PT := T#10S);
    END_IF
END_IF

IF new_check THEN	
	GVL.healthy_inv := 0;
	FOR i := 1 TO GVL.n_slave DO
		//i := 1;
		IF GVL.inv[i].write_done THEN
	
			CASE GVL.inv[i].read_state OF
			
				0:
					check_inverter_health[i](
						sIPAddr:= GVL.server_addr, 
						nTCPPort:= GVL.inv[i].tcp_port, 
						nUnitID:= GVL.inv[i].unit_id, 
						nQuantity:= GVL.inv[i].health, 
						nMBAddr:= GVL.inv[i].mb_h_addr, 
						cbLength:= SIZEOF(GVL.inv[i].health), 
						pDestAddr:= ADR(GVL.inv[i].health), 
						bExecute:= TRUE, 
						tTimeout:= T#2S, 
						bBusy=> , 
						bError=> , 
						nErrId=> , 
						cbRead=> 
					);
					GVL.inv[i].read_state := 1;
					
				
				// TO DO aggiungi un counter e un limite superato il quale stabilisci che l'inverter non funziona
				1:
					check_inverter_health[i](bExecute := FALSE);
					IF NOT check_inverter_health[i].bBusy THEN
						IF check_inverter_health[i].bError THEN 
							GVL.inv[i].health := 0;
						END_IF
						GVL.inv[i].read_state := 0;
						GVL.inv[i].read_done := TRUE; 
					END_IF
					
					IF GVL.inv[i].health = 1 THEN
						GVL.healthy_inv := GVL.healthy_inv + 1; 
					END_IF
				
			END_CASE
			
		END_IF
		
	END_FOR
	
//ELSE
//	GVL.healthy_inv := 0; 
//	FOR i := 1 TO GVL.n_slave DO
//		IF GVL.inv[i].health = 1 THEN
//			GVL.inv[i].read_done := TRUE;
//			GVL.healthy_inv := GVL.healthy_inv + 1;
//		END_IF	
//	END_FOR
//END_IF

all_done := TRUE; // all_done è una variabile booleana dichiarata in precedenza
    FOR i := 1 TO GVL.n_slave DO
        IF NOT GVL.inv[i].read_done THEN
            all_done := FALSE;
        END_IF;
    END_FOR;
    
    // Se tutte le letture sono finite, si resetta new_check per preparare il prossimo ciclo
    IF all_done THEN
        new_check := FALSE;
        // (Opzionale) Reset dello stato di lettura di ciascun inverter per il prossimo ciclo
        FOR i := 1 TO GVL.n_slave DO
            GVL.inv[i].read_done := FALSE;
        END_FOR;
    END_IF;
END_IF;

END_FUNCTION_BLOCK

// ---- POUs/Programs/Algorithms/Active power regulation/Active_Power_Regulation.TcPOU
FUNCTION_BLOCK Active_Power_Regulation
VAR_INPUT
END_VAR
VAR_OUTPUT
END_VAR
VAR
	i: UINT;
	difference: REAL;
	update_pi_sp: FB_PI_Setpoint;
	timer_sp: TON;
	temp_sp: REAL;
	reach_sp: FB_Reach_SP_ActP;
	act_pwr_freq_reg_sp: FB_Frequency_Regulation;
END_VAR

IF GVL.WISNAM_PPC.active_power_ctrl_enabled THEN
	
	/// 1. MULTI-INPUT REDUCER + 4. NORMALIZATION ACTIVE POWER ///////////////////////////////////////	
	temp_sp := sp_input_reducer(sp_auto := GVL_Act_Pwr.setpoint_auto, sp_manual := GVL_Act_Pwr.setpoint_manual, sp_tso := GVL_Act_Pwr.setpoint_tso); 
	IF temp_sp <> GVL_Act_Pwr.setpoint_mem THEN
		GVL_Act_Pwr.setpoint := low_pass_filter(plant_target := temp_sp, filter_output_mem := GVL_Act_Pwr.setpoint_mem, alpha := GVL.plant_sp_alpha);
		GVL_Act_Pwr.target_prod := GVL_Act_Pwr.setpoint * GVL.power_plant.nominal_power;
	
		IF NOT GVL_Act_Pwr.ramp_rate_follow_inv THEN
			GVL_Act_Pwr.ramp_rate_follow_inv := TRUE;
		END_IF
					
		IF NOT GVL_Act_Pwr.ramp_rate_ctrl THEN
			GVL_Act_Pwr.ramp_rate_ctrl := TRUE;
		END_IF 	
			
	END_IF
		
	/// 6. CONTROL ACTIVE POWER-FREQUENCY //////////////////////////////////////////	
	GVL_Freq.frequency_smoothed := low_pass_filter(plant_target := GVL.VIRTUAL_METER.frequency, filter_output_mem := GVL_Freq.frequency_smoothed_mem, alpha := GVL_Act_Pwr.setpoint_alpha); // TO DO: valuta se imppostare alpha a 1
	GVL_Freq.frequency_smoothed_mem := GVL_Freq.frequency_smoothed;
	GVL_Freq.p_nd := 0;
	
	FOR i := 1 TO GVL.n_slave DO
		IF GVL.inv[i].health = 1 THEN
			GVL_Freq.p_nd := GVL_Freq.p_nd + GVL.inv[i].active_pwr_nominal_pwr;
		END_IF
	END_FOR
	
	GVL_Freq.p_nd := GVL_Freq.p_nd / GVL.power_plant.nominal_power;
	
	IF GVL.WISNAM_PPC.actp_freq_reg_enabled THEN
		
//		GVL_Freq.output_pf_regulation := deltaActivePwr_Frequency_Regulation(
//									p_nd := GVL_Freq.p_nd, 	// scelta corretta ?? 
//									current_frequency := GVL_Freq.frequency_smoothed, 
//									current_power := GVL.VIRTUAL_METER.active_power_sp
//									//pe_selector := TO_INT(0) // nella versione di codice cui ho accesso, la variabile "underFreqDropDynamicRef" è posta = 0
//									);
//		act_pwr_freq_reg_sp(current_power := GVL.VIRTUAL_METER.active_power_prod, 
//							current_frequency := GVL.VIRTUAL_METER.frequency,
//							p_nd := GVL_Freq.p_nd,
//							target_pfn => GVL_Freq.prod_nominal_freq
//							);
							
	END_IF
	
	
	/// 8. TARGET LIMITER (da rivedere)//////////	
	IF (GVL_Act_Pwr.total_sp < 0) THEN
		GVL_Act_Pwr.total_sp := 0;
	ELSIF  (GVL_Act_Pwr.total_sp > 1) THEN
		GVL_Act_Pwr.total_sp := 1;
	END_IF
	
	/// minimum step size: 5% ///
	IF (GVL_Act_Pwr.setpoint_mem = 0 AND (GVL_Act_Pwr.total_sp > 0 AND GVL_Act_Pwr.total_sp < 0.05)) THEN
		GVL_Act_Pwr.total_sp := 0.05;
	END_IF
	
	IF (GVL_Act_Pwr.total_sp < 0.05 AND GVL_Act_Pwr.setpoint_mem >= 0.05) THEN
		GVL_Act_Pwr.total_sp := 0;
	END_IF
	
//	difference := GVL_Act_Pwr.setpoint - GVL_Act_Pwr.setpoint_mem; 
//	IF ABS(difference) > GVL.power_plant_max_sp_increase AND GVL_Act_Pwr.ramp_rate_ctrl THEN
//		IF difference > 0 THEN	
//			GVL_Act_Pwr.setpoint := GVL_Act_Pwr.setpoint_mem + GVL.power_plant_max_sp_increase;
//		ELSE
//			GVL_Act_Pwr.setpoint := GVL_Act_Pwr.setpoint_mem - GVL.power_plant_max_sp_increase;
//		END_IF
//	END_IF
	
	GVL_Act_Pwr.setpoint_mem := GVL_Act_Pwr.setpoint;
	reach_sp(sp_target_actp := GVL_Act_Pwr.setpoint); 	

END_IF

END_FUNCTION_BLOCK

// ---- POUs/Programs/Algorithms/Active power regulation/FB_Frequency_Regulation.TcPOU
FUNCTION_BLOCK FB_Frequency_Regulation
VAR_INPUT
	current_power: REAL;
	current_frequency: REAL;
	p_nd: REAL;
END_VAR
VAR_OUTPUT
	target_pfn: REAL;
END_VAR
VAR
	f_error: REAL;
	power_percentage_delta: REAL;
	overshoot_freq_error: REAL;
	delta_p: REAL;
	available_power: REAL;
END_VAR

available_power := p_nd * GVL.power_plant.nominal_power;
target_pfn := current_power;

/// dead-band ////////////////////////////////////////////
IF GVL_Freq.under_f_db_threshold <= current_frequency AND current_frequency <= GVL_Freq.over_f_db_threshold THEN
	GVL_Freq.frequency_regulation_priority := FALSE;	
	RETURN;
END_IF
/////////////////////////////////////////////////////////

/// critical scenarios /////////////////////////////////
IF current_frequency > GVL_Freq.max_value_over_f THEN
	target_pfn := 0;
	GVL_Freq.frequency_regulation_priority := TRUE;
	RETURN;
END_IF


IF current_frequency < GVL_Freq.min_value_under_f THEN
	target_pfn := p_nd;
	GVL_Freq.frequency_regulation_priority := TRUE;
	RETURN;
END_IF
/////////////////////////////////////////////////////////


/// FSM-O ///////////////////////////////////////////////
IF GVL_Freq.over_f_db_threshold < current_frequency AND current_frequency <= GVL_Freq.over_f_medium_threshold THEN
	GVL_Freq.frequency_regulation_priority := TRUE;
	f_error := ABS(current_frequency - GVL_Freq.frequency_reference);
	power_percentage_delta := f_error*GVL_Freq.S_over_mid_val;
END_IF
/////////////////////////////////////////////////////////


/// FSM-U ///////////////////////////////////////////////
IF GVL_Freq.under_f_db_threshold > current_frequency AND current_frequency >= GVL_Freq.under_f_medium_threshold THEN
	GVL_Freq.frequency_regulation_priority := TRUE;
	f_error := ABS(current_frequency - GVL_Freq.frequency_reference);
	power_percentage_delta := f_error*GVL_Freq.S_under_mid_val;
END_IF
/////////////////////////////////////////////////////////


/// LFSM-O //////////////////////////////////////////////
IF GVL_Freq.over_f_medium_threshold < current_frequency THEN
	GVL_Freq.frequency_regulation_priority := TRUE;
	f_error := ABS(current_frequency - GVL_Freq.frequency_reference);
	overshoot_freq_error := ABS(GVL_Freq.over_f_medium_threshold - GVL_Freq.over_f_db_threshold)/20; // TO DO: parametrizzare
	power_percentage_delta := (f_error + overshoot_freq_error)*GVL_Freq.S_over_ext_val;
END_IF
/////////////////////////////////////////////////////////


/// LFSM-U //////////////////////////////////////////////
IF GVL_Freq.under_f_medium_threshold > current_frequency THEN
	GVL_Freq.frequency_regulation_priority := TRUE;
	f_error := ABS(current_frequency - GVL_Freq.frequency_reference);
	overshoot_freq_error := ABS(GVL_Freq.under_f_medium_threshold - GVL_Freq.under_f_db_threshold)/20; // TO DO: parametrizzare
	power_percentage_delta := (f_error + overshoot_freq_error)*GVL_Freq.S_over_ext_val;	
END_IF
/////////////////////////////////////////////////////////

delta_p := (available_power/100) * power_percentage_delta;
IF current_frequency > GVL_Freq.frequency_reference THEN
	target_pfn := current_power - delta_p;
ELSE
	target_pfn := current_power + delta_p;
END_IF

END_FUNCTION_BLOCK

// ---- POUs/Programs/Algorithms/sp_input_reducer.TcPOU
FUNCTION sp_input_reducer : real
VAR_INPUT
	sp_auto: REAL;
	sp_manual: REAL;
	sp_tso: REAL;
END_VAR
VAR
END_VAR

sp_input_reducer := 1;

IF GVL.WISNAM_PPC.REMOTE_MODE THEN
	sp_input_reducer := sp_tso;
END_IF


IF GVL.WISNAM_PPC.AUTO_MODE THEN
	IF sp_input_reducer > sp_auto THEN
		sp_input_reducer := sp_auto;
	END_IF
END_IF


IF GVL.WISNAM_PPC.MANUAL_MODE THEN
	IF sp_input_reducer > sp_manual THEN
		sp_input_reducer := sp_manual;
	END_IF
END_IF

END_FUNCTION

// ---- POUs/Programs/Algorithms/Reactive power regulation/Reactive_Power_Regulation.TcPOU
FUNCTION_BLOCK Reactive_Power_Regulation
VAR_INPUT
END_VAR
VAR_OUTPUT
END_VAR
VAR
	difference: REAL;
	update_pi_sp_q: FB_PI_Setpoint;
	i: UINT;
	norm_error_mem: REAL;
	react_pwr_voltage_ctrl: FB_ReactivePwr_Voltage_Ctrl;
	reach_sp: FB_Reach_SP_ReactP;
	temp_sp: REAL;
END_VAR

IF GVL.WISNAM_PPC.reactive_power_ctrl_enabled OR GVL.WISNAM_PPC.power_factor_ctrl_enabled THEN
	
	IF NOT GVL.WISNAM_PPC.power_factor_ctrl_enabled THEN
		temp_sp := sp_input_reducer(sp_auto := GVL_React_Pwr.setpoint_auto, sp_manual := GVL_React_Pwr.setpoint_manual, sp_tso := GVL_React_Pwr.setpoint_tso);
		IF temp_sp <> GVL_React_Pwr.setpoint_mem THEN
			GVL_React_Pwr.setpoint := Low_Pass_Filter(plant_target := temp_sp, filter_output_mem := GVL_React_Pwr.setpoint_mem, alpha := GVL.plant_sp_alpha); 
			GVL_React_Pwr.target_prod := GVL_React_Pwr.setpoint * GVL.power_plant.nominal_power;
		END_IF
	END_IF
	
	/// controllo potenza reattiva - tensione ///
	IF GVL.WISNAM_PPC.qv_ctrl_enabled THEN
		GVL_React_Pwr.p_nd := 0;
		FOR i := 1 TO GVL.n_slave DO
			IF GVL.inv[i].health = 1 THEN
				GVL_React_Pwr.p_nd := GVL_React_Pwr.p_nd + GVL.inv[i].active_pwr_nominal_pwr;
			END_IF
		END_FOR
		GVL_React_Pwr.p_nd := GVL_React_Pwr.p_nd / GVL.power_plant.nominal_power;
	
		GVL_Voltage.v_norm := GVL.VIRTUAL_METER.measured_voltage / GVL_Voltage.reference_value; // PLOT
		GVL_Voltage.error := GVL.VIRTUAL_METER.measured_voltage - GVL_Voltage.reference_value; 
		GVL_Voltage.norm_error := GVL_Voltage.error / GVL_Voltage.reference_value;
		GVL_Voltage.norm_error := Low_Pass_Filter(plant_target := GVL_Voltage.norm_error, filter_output_mem := norm_error_mem, alpha := GVL_React_Pwr.setpoint_alpha);
		norm_error_mem := GVL_Voltage.norm_error; 
		
		react_pwr_voltage_ctrl();
	ELSE
		GVL_Voltage.output_qv_regulation := 0;
	END_IF	
	
	
	
//	IF GVL.WISNAM_PPC.power_factor_ctrl_enabled THEN
		
//		GVL_React_Pwr.target_prod := TO_REAL((GVL.VIRTUAL_METER.active_power_prod / GVL_React_Pwr.power_factor_target) * SQRT(1 - EXPT(GVL_React_Pwr.power_factor_target,2)));
//		GVL_React_Pwr.setpoint := GVL_React_Pwr.target_prod / GVL.power_plant.nominal_power;
		
//	END_IF
	
	
	/// 8. PLANT TARGET (chiedi Carmelo)/// 
	GVL_React_Pwr.total_sp := GVL_React_Pwr.setpoint + GVL_Voltage.output_qv_regulation;
	
	IF GVL_React_Pwr.total_sp > GVL_React_Pwr.max_q_pf_regulation AND GVL.WISNAM_PPC.power_factor_ctrl_enabled THEN
		
		GVL_React_Pwr.total_sp := GVL_React_Pwr.max_q_pf_regulation;
	
	END_IF
	
	
	IF (GVL_React_Pwr.setpoint < 0) OR (GVL_React_Pwr.setpoint > GVL.power_plant_max_sp_q) THEN
		GVL_React_Pwr.setpoint := GVL_React_Pwr.setpoint_mem;
	END_IF
	
	/// minimum step size: 5% ///
	IF (GVL_React_Pwr.setpoint_mem = 0 AND (GVL_React_Pwr.setpoint > 0 AND GVL_React_Pwr.setpoint < 0.05)) THEN
		GVL_React_Pwr.setpoint := 0.05;
	END_IF
	
	IF (GVL_React_Pwr.setpoint < 0.05 AND GVL_React_Pwr.setpoint_mem >= 0.05) THEN
		GVL_React_Pwr.setpoint := 0;
	END_IF
	
	
//	difference := GVL_React_Pwr.setpoint - GVL_React_Pwr.setpoint_mem; 
//	IF ABS(difference) > GVL.power_plant_max_sp_increase_q THEN
//		IF difference > 0 THEN	
//			GVL_React_Pwr.setpoint := GVL_React_Pwr.setpoint_mem + GVL.power_plant_max_sp_increase_q;
//		ELSE
//			GVL_React_Pwr.setpoint := GVL_React_Pwr.setpoint_mem - GVL.power_plant_max_sp_increase_q;
//		END_IF
//	END_IF
//	GVL_React_Pwr.setpoint_mem := GVL_React_Pwr.setpoint;
	
	GVL_React_Pwr.setpoint_mem := GVL_React_Pwr.setpoint;	

	reach_sp(sp_target_reactp := GVL_React_Pwr.total_sp);
	

END_IF

END_FUNCTION_BLOCK

// ---- POUs/Programs/Algorithms/Reactive power regulation/FB_ReactivePwr_Voltage_Ctrl.TcPOU
FUNCTION_BLOCK FB_ReactivePwr_Voltage_Ctrl
VAR_INPUT
END_VAR
VAR_OUTPUT
END_VAR
VAR
	fbCTRL_PI: FB_CTRL_PI;
	stCTRL_PI_PARAMS: ST_CTRL_PI_PARAMS;
	eMode: E_CTRL_MODE;
	bInit: BOOL := TRUE;
	fbTON: TON;
	hysteresis_block: FB_Hysteresis;
	map_QV: FB_Map_QV;
END_VAR

IF bInit THEN
	(* init parameter struct *)
	stCTRL_PI_PARAMS.tCtrlCycleTime		:= T#50MS;
	stCTRL_PI_PARAMS.tTaskCycleTime		:= T#10MS;
	stCTRL_PI_PARAMS.tTn				:= T#2000MS;		(* integral gain Tn				*)
	stCTRL_PI_PARAMS.fKp				:= 0.04;			(* proportional gain Kp				*)
	stCTRL_PI_PARAMS.fOutMaxLimit		:= GVL_Voltage.pi_ctrl_max_output;  		(* maximum output limit				*)
	stCTRL_PI_PARAMS.fOutMinLimit		:= GVL_Voltage.pi_ctrl_min_output;			(* minimum output limit				*)

	(* set the mode to ACTIVE --> normal operation *)
	eMode := eCTRL_MODE_ACTIVE;

	(* reset the init flag *)
	bInit := FALSE;
END_IF


fbCTRL_PI(
	fSetpointValue:= 0, 
	fActualValue:= GVL_Voltage.norm_error, 
	fManSyncValue:= , 
	bSync:= , 
	eMode:= eMode, 
	bHold:= , 
	fOut=> GVL_Voltage.output_pi, 
	bARWactive=> , 
	eState=> , 
	eErrorId=> , 
	bError=> , 
	stParams:= stCTRL_PI_PARAMS
	);

/// TO DO: dopo che avremo definito gli schemi di controllo, mettere i PID in una FB separata.
	
/// REGULATOR LIMITER /////////////////////////////////////////////////////// 
//IF GVL_Voltage.output_pi > GVL_Voltage.max_norm_correction THEN
//	GVL_Voltage.output_pi := GVL_Voltage.max_pi_correction;
//ELSIF GVL_Voltage.output_pi < GVL_Voltage.min_pi_correction THEN
//	GVL_Voltage.output_pi := GVL_Voltage.min_norm_correction;
//END_IF
/////////////////////////////////////////////////////////////////////////////

/// HYSTERESIS ////////////////////////////////////////////////////////////// 
hysteresis_block();
/////////////////////////////////////////////////////////////////////////////

/// Q/V MAP /////////////////////////////////////////////////////////////////
map_QV();
/////////////////////////////////////////////////////////////////////////////

//GVL_Voltage.output_qv_regulation := deltaReactivePwr_Voltage_Regulation(input := GVL_Voltage.output_qv_regulation);

GVL_Voltage.output_qv_regulation := GVL_Voltage.output_qv_regulation * GVL_React_Pwr.p_nd;

/// LIMITATORE GLOBALE DEL REGOLATORE ///////////////////////////////////////
IF GVL_Voltage.output_qv_regulation > 0.3 THEN	// TO DO: assicurati che questi dati siano giusti 
	GVL_Voltage.output_qv_regulation := 0.3;
ELSIF GVL_Voltage.output_qv_regulation < -0.35 THEN
	GVL_Voltage.output_qv_regulation := -0.35;
END_IF
/////////////////////////////////////////////////////////////////////////////

END_FUNCTION_BLOCK

// ---- POUs/Programs/Algorithms/Reactive power regulation/FB_Hysteresis.TcPOU
FUNCTION_BLOCK FB_Hysteresis
VAR_INPUT
END_VAR
VAR_OUTPUT
END_VAR
VAR
	half_clearance: REAL;
	cap: REAL;
	floor: REAL;
END_VAR

half_clearance := GVL_Voltage.hyst_clearance / 2;
cap := GVL_Voltage.output_pi + half_clearance;
floor := GVL_Voltage.output_pi - half_clearance;

GVL_Voltage.output_qv_regulation := MIN(cap, MAX(floor, GVL_Voltage.last_output_qv_regulation));
GVL_Voltage.last_output_qv_regulation := GVL_Voltage.output_qv_regulation;

END_FUNCTION_BLOCK

// ---- POUs/Programs/Algorithms/Reactive power regulation/FB_Map_QV.TcPOU
FUNCTION_BLOCK FB_Map_QV
VAR_INPUT
END_VAR
VAR_OUTPUT
END_VAR
VAR
	A: stQV_POINT;
	B: stQV_POINT;
	C: stQV_POINT;
	D: stQV_POINT;
	E: stQV_POINT;
	F: stQV_POINT;
	G: stQV_POINT;
	
	max_qv_correction: REAL;
	min_qv_correction: REAL;
	v_ratio: REAL;
	t: REAL;
	i: UINT;
	x: REAL;
	y: REAL;
END_VAR

v_ratio := GVL.VIRTUAL_METER.measured_voltage / GVL_Voltage.reference_value;

/// definizione delle coordiante dei punti della mappa Q/V///
A.q_pnd_ratio := 0;
A.voltage_ratio := 1.1;

B.q_pnd_ratio := 0.30;
B.voltage_ratio := 1.05;

C.q_pnd_ratio := 0.30;
C.voltage_ratio := 0.95;

D.q_pnd_ratio := 0;
D.voltage_ratio := 0.9;

E.q_pnd_ratio := -0.35;
E.voltage_ratio := 0;
/////////////////////////////////////////////////////////////

IF v_ratio > B.voltage_ratio AND v_ratio <= A.voltage_ratio THEN
	min_qv_correction := -0.35;
	t := (v_ratio - A.voltage_ratio) / (A.voltage_ratio - B.voltage_ratio);
	max_qv_correction := t*B.q_pnd_ratio + (1 - t)*A.q_pnd_ratio;
 


ELSIF v_ratio <= B.voltage_ratio AND v_ratio >= C.voltage_ratio THEN
	max_qv_correction := 0.30;
	min_qv_correction := -0.35;



ELSIF v_ratio < C.voltage_ratio AND v_ratio >= D.voltage_ratio THEN
	max_qv_correction := 0.30;
	t := (v_ratio - D.voltage_ratio) / (C.voltage_ratio - D.voltage_ratio);
	min_qv_correction := t*C.q_pnd_ratio + (1 - t)*D.q_pnd_ratio; 
END_IF 


// TO DO: per implementazioni future di una regolazione mediante mappa 
//FOR i := 1 TO GVL_React_Pwr.n_points DO
//	IF v_ratio >= GVL_React_Pwr.enhanced_points[i][1] THEN 
//		x := GVL_React_Pwr.enhanced_points[i][1];
//		y := GVL_React_Pwr.enhanced_points[i][2];
//		g := GVL_React_Pwr.enhanced_points[i][3];
		
//		GVL_Voltage.output_qv_regulation := y + g*(v_ratio - x);
//		EXIT
//	END_IF
//END_FOR


IF GVL_Voltage.output_qv_regulation < min_qv_correction THEN
	GVL_Voltage.output_qv_regulation := min_qv_correction;
END_IF
	
IF GVL_Voltage.output_qv_regulation > max_qv_correction THEN
	GVL_Voltage.output_qv_regulation := max_qv_correction;
END_IF

END_FUNCTION_BLOCK

// ---- POUs/Programs/Algorithms/Reactive power regulation/FB_Reach_SP_ReactP.TcPOU
FUNCTION_BLOCK FB_Reach_SP_ReactP
VAR_INPUT
	sp_target_reactp: REAL;
END_VAR
VAR_OUTPUT
END_VAR
VAR
	setpoint_to_send_ff: REAL;
	filtered_sp: REAL;
	update_pi_sp: FB_PI_Setpoint;
	low_pass_filter_mem: REAL;
	pi_correction: REAL;
END_VAR

IF ABS(GVL.VIRTUAL_METER.reactive_power_sp - sp_target_reactp) > GVL_React_Pwr.sp_tolerance_q THEN
		
		IF GVL_React_Pwr.ff_pi_q_control_enable THEN

			/// 10. PREACTION FF ///
			setpoint_to_send_ff := FF_BLOCK(input_value := sp_target_reactp, k_ff := 0.025);
			
			/// 9. LOW PASS FILTER + 12. FEEDBACK ///
			filtered_sp := Low_Pass_Filter(plant_target := sp_target_reactp, filter_output_mem := low_pass_filter_mem_q, alpha := GVL_React_Pwr.setpoint_alpha);
			low_pass_filter_mem_q := filtered_sp;
		
			update_pi_sp_q(sp_value := GVL_React_Pwr.filtered_setpoint, feedback_sp := GVL.VIRTUAL_METER.reactive_power_sp, pi_output => GVL_React_Pwr.pi_correction_q);
			
			/// 13. TOTAL PLANT COMMAND ///
			GVL_React_Pwr.setpoint_to_send := setpoint_to_send_ff + pi_correction_q;
			GVL_React_Pwr.expected_pod_prod_q := GVL_React_Pwr.setpoint_to_send * GVL.power_plant.nominal_power;

		ELSE
			
			CASE GVL_React_Pwr.reactive_pwr_ctrl_case OF
				1: 
					// update setpoint
					GVL_React_Pwr.setpoint_to_send := GVL_React_Pwr.setpoint_alpha * sp_target_reactp + (1-GVL_React_Pwr.setpoint_alpha) * GVL.VIRTUAL_METER.reactive_power_sp;
					GVL_React_Pwr.expected_pod_prod_q := GVL_React_Pwr.setpoint_to_send*GVL.power_plant.nominal_power;
					GVL_React_Pwr.reactive_pwr_ctrl_case := 2;
				2:
					// wait until the plant is close to current setpoint
					IF ABS(GVL_React_Pwr.setpoint_to_send - GVL.VIRTUAL_METER.reactive_power_sp) < 0.1 THEN
						GVL_React_Pwr.reactive_pwr_ctrl_case := 1;
					END_IF
				3:
					// fault management
			END_CASE  
	   END_IF
	   
	   IF GVL_React_Pwr.expected_pod_prod_q > GVL.power_plant.nominal_power THEN
			GVL_React_Pwr.setpoint_to_send := 1;
			GVL_React_Pwr.expected_pod_prod_q := GVL.power_plant.nominal_power;
		END_IF
	   
	END_IF

END_FUNCTION_BLOCK

// ---- POUs/Programs/Engine/MQTT_TSO_Comm.TcPOU
FUNCTION_BLOCK MQTT_TSO_Comm
VAR_OUTPUT
END_VAR
VAR
	init_mqtt: BOOL := TRUE;
	mqtt_client: FB_IotMqttClient;
	message_queue: FB_IotMqttMessageQueue;
	message: FB_IotMqttMessage;
	
	subscribed_act_pwr: BOOL;
	topic_act_pwr: STRING(255) := 'act_p_setpoint/topic';
	receiving_topic_act_pwr: STRING(255);
	receiving_data_act_pwr: STRING(255);
	
	subscribed_react_pwr: BOOL;
	topic_react_pwr: STRING(255) := 'react_p_setpoint/topic';
	receiving_topic_react_pwr: STRING(255);
	receiving_data_react_pwr: STRING(255);
	
	receiving_topic: STRING(255);
	receiving_data: STRING(255);
END_VAR

IF init_mqtt THEN
	mqtt_client.sHostName := 'localhost';
	mqtt_client.nHostPort := 1883;
	mqtt_client.sTopicPrefix := '';
	mqtt_client.ipMessageQueue := message_queue;
	mqtt_client.sClientId := 'TSO';
	
	init_mqtt := FALSE;
END_IF

mqtt_client.Execute(bConnect := TRUE);

IF mqtt_client.bConnected THEN
	IF NOT subscribed_act_pwr AND GVL.WISNAM_PPC.active_power_ctrl_enabled THEN
		subscribed_act_pwr := mqtt_client.Subscribe(sTopic := topic_act_pwr, eQoS := TcIotMqttQos.AtMostOnceDelivery);
	END_IF
	
	IF NOT subscribed_react_pwr AND GVL.WISNAM_PPC.reactive_power_ctrl_enabled THEN
		subscribed_react_pwr := mqtt_client.Subscribe(sTopic := topic_react_pwr, eQoS := TcIotMqttQos.AtMostOnceDelivery);
	END_IF
END_IF

IF message_queue.nQueuedMessages > 0 THEN
	IF message_queue.Dequeue(fbMessage := message) THEN
		message.GetTopic(pTopic := ADR(receiving_topic), nTopicSize := SIZEOF(receiving_topic));	
		message.GetPayload(pPayload := ADR(receiving_data), nPayloadSize := SIZEOF(receiving_data), bSetNullTermination := FALSE);
		
		IF receiving_topic = 'act_p_setpoint/topic' THEN
			GVL_Act_Pwr.setpoint_tso := setpoint_acquired(message_received := receiving_data);
		ELSIF receiving_topic = 'react_p_setpoint/topic' THEN 
			GVL_React_Pwr.setpoint_tso := setpoint_acquired(message_received := receiving_data);
		END_IF

	END_IF
END_IF

END_FUNCTION_BLOCK

// ---- POUs/Programs/Algorithms/setpoint_acquired.TcPOU
FUNCTION setpoint_acquired : REAL
VAR_INPUT
	message_received: STRING(255);
END_VAR
VAR
	aux_string_array: ARRAY[1..GVL.max_message_info] OF STRING(255);
	split_mqtt_message: BOOL;
	j: UINT;
END_VAR

aux_string_array[1] := message_received;
FOR j := 1 TO GVL.max_message_info - 1 DO
	split_mqtt_message := FindAndSPlitChar(
										sSeparatorChar := ':',
										pSrcString := ADR(aux_string_array[j]),
										pLeftString := ADR(aux_string_array[j]),
										nLeftSize := SIZEOF(aux_string_array[j]),
										pRightString := ADR(aux_string_array[j + 1]), 
										nRightSize := SIZEOF(aux_string_array[j + 1]),
										bSearchFromRight := FALSE
										);
END_FOR
setpoint_acquired := STRING_TO_REAL(aux_string_array[2]);

END_FUNCTION

// ---- POUs/Programs/Algorithms/Load Following/FB_Load_Following.TcPOU
FUNCTION_BLOCK FB_Load_Following
VAR_INPUT
END_VAR
VAR_OUTPUT
END_VAR
VAR
	i: UINT;
	error_perc: REAL;
	delta: REAL; 
	reach_sp: FB_Reach_SP_ActP;
END_VAR

//  TO DO: valutare se, nel caso della potenza erogata dalla rete, conviene esprimere la potenza in termini percentuali rispetto alla potenza di rete
error_perc := ((GVL.VIRTUAL_POI_METER.active_power_prod - GVL_Load_Following.power_grid_max) / GVL_Load_Following.power_grid_max) * 100;

IF GVL.VIRTUAL_POI_METER.active_power_prod <= GVL_Load_Following.power_grid_min THEN
	
	delta := 0;
	GVL_Act_Pwr.total_sp := 0;

ELSIF (GVL.VIRTUAL_POI_METER.active_power_prod >= GVL_Load_Following.power_grid_min) AND (GVL.VIRTUAL_POI_METER.active_power_prod <= GVL_Load_Following.power_grid_max) THEN 
	
	delta := -1 *GVL_Load_Following.delta_fast;

ELSE

	delta := GVL_Load_Following.delta_fast;	

END_IF


IF (error_perc > 10) AND (error_perc < GVL_Load_Following.max_error_perc) THEN
	
	delta := GVL_Load_Following.delta_slow;

END_IF


IF error_perc < 10 THEN
	
	delta := 0;

END_IF

// TO DO: verificare se questa formula è corretta
GVL_Act_Pwr.total_sp := GVL_Act_Pwr.total_sp + delta * 0.100;   // + delta * dT con dT = tempo di esecuzione del main, pari a 100ms	
GVL_Act_Pwr.total_sp := MAX(0, MIN(1, GVL_Act_Pwr.total_sp)); 

reach_sp(sp_target_actp := GVL_Act_Pwr.total_sp);

END_FUNCTION_BLOCK

// ---- POUs/Programs/Algorithms/Meter/Update_Virtual_Meter.TcPOU
FUNCTION Update_Virtual_Meter : bool
VAR_INPUT
END_VAR
VAR
	i: UINT;
END_VAR

GVL.VIRTUAL_METER.active_power_prod := 0;
GVL.VIRTUAL_METER.reactive_power_prod := 0;
GVL.VIRTUAL_METER.frequency := 0;
GVL.VIRTUAL_METER.measured_voltage := 0;

GVL.VIRTUAL_POI_METER.active_power_prod := 0;
GVL.VIRTUAL_POI_METER.reactive_power_prod := 0;
GVL.VIRTUAL_POI_METER.frequency := 0;
GVL.VIRTUAL_POI_METER.measured_voltage := 0;

FOR i := 1 TO GVL.n_meter DO
	
	IF GVL.meter_arr[i].pos = stGRID_POS.pu THEN
		
		GVL.VIRTUAL_METER.active_power_prod := GVL.VIRTUAL_METER.active_power_prod + GVL.meter_arr[i].active_power_prod;
		GVL.VIRTUAL_METER.reactive_power_prod := GVL.VIRTUAL_METER.reactive_power_prod + GVL.meter_arr[i].reactive_power_prod;
		GVL.VIRTUAL_METER.frequency	:= GVL.VIRTUAL_METER.frequency + GVL.meter_arr[i].frequency;
		GVL.VIRTUAL_METER.measured_voltage := GVL.VIRTUAL_METER.measured_voltage + GVL.meter_arr[i].measured_voltage;
		
	ELSE
		
		GVL.VIRTUAL_POI_METER.active_power_prod := GVL.VIRTUAL_POI_METER.active_power_prod + GVL.meter_arr[i].active_power_prod;
		GVL.VIRTUAL_POI_METER.reactive_power_prod := GVL.VIRTUAL_POI_METER.reactive_power_prod + GVL.meter_arr[i].reactive_power_prod;
		GVL.VIRTUAL_POI_METER.frequency	:= GVL.VIRTUAL_POI_METER.frequency + GVL.meter_arr[i].frequency;
		GVL.VIRTUAL_POI_METER.measured_voltage := GVL.VIRTUAL_POI_METER.measured_voltage + GVL.meter_arr[i].measured_voltage;	
	
	END_IF
	
END_FOR

GVL.VIRTUAL_METER.frequency := GVL.VIRTUAL_METER.frequency / GVL.n_meter_pu;
GVL.VIRTUAL_METER.measured_voltage := GVL.VIRTUAL_METER.measured_voltage / GVL.n_meter_pu;
GVL.VIRTUAL_METER.active_power_sp := GVL.VIRTUAL_METER.active_power_prod / GVL.power_plant.nominal_power;
GVL.VIRTUAL_METER.reactive_power_sp := GVL.VIRTUAL_METER.reactive_power_prod / GVL.power_plant.nominal_power; 

GVL.VIRTUAL_POI_METER.frequency := GVL.VIRTUAL_POI_METER.frequency / GVL.n_meter_poi;
GVL.VIRTUAL_POI_METER.measured_voltage := GVL.VIRTUAL_POI_METER.measured_voltage / GVL.n_meter_poi;
GVL.VIRTUAL_POI_METER.active_power_sp := GVL.VIRTUAL_POI_METER.active_power_prod / GVL.power_plant.nominal_power;
GVL.VIRTUAL_POI_METER.reactive_power_sp := GVL.VIRTUAL_POI_METER.reactive_power_prod / GVL.power_plant.nominal_power;

END_FUNCTION

// ---- POUs/Programs/Engine/Inverter Comm/FB_Comm_Setup.TcPOU
FUNCTION_BLOCK FB_Comm_Setup
VAR_INPUT
END_VAR
VAR_OUTPUT
END_VAR
VAR
	start: BOOL;
	i: UINT;
END_VAR

/// INIT PLANT PARAMETERS ///////////////////////////
FOR i := 1 TO GVL.n_slave DO
	/// server info ///
	GVL.inv[i].tcp_port := GVL.initial_tcp_port + i;	
	GVL.inv[i].unit_id := 1;
	
	/// active power ///
	GVL.inv[i].n_quantity_act_pwr := 2;
	GVL.inv[i].mb_addr_act_pwr := 1;
	GVL.inv[i].active_pwr_nominal_pwr := GVL.power_plant.nominal_power / Gvl.n_slave;
	
	/// inverter status /// 
	GVL.inv[i].health := 1;
	GVL.inv[i].mb_h_addr := 0;
	GVL.inv[i].health_quantity := 1;
	
	/// reactive power ///
	GVL.inv[i].n_quantity_react_pwr := 2;
	GVL.inv[i].mb_addr_react_pwr := 3;
	GVL.inv[i].reactive_pwr_nominal_pwr := GVL.power_plant.nominal_power / GVL.n_slave;
	
	/// init set point memory ////
	GVL_Act_Pwr.setpoint_mem := GVL_Act_Pwr.setpoint;
	GVL_React_Pwr.setpoint_mem := GVL_React_Pwr.setpoint;
END_FOR

END_FUNCTION_BLOCK

// ---- POUs/Programs/Engine/FB_Setup_Meter_Comm.TcPOU
FUNCTION_BLOCK FB_Setup_Meter_Comm
VAR_INPUT
END_VAR
VAR_OUTPUT
END_VAR
VAR
	 i: UINT;
END_VAR

FOR i:= 1 TO GVL.n_meter DO
	GVL.meter_arr[i].tcp_port := 9501 - (i - 1);
	GVL.meter_arr[i].unit_id := 1;
	
	GVL.meter_arr[i].nQuantity_Act_Pwr := 4;
	GVL.meter_arr[i].nMBAddr_Act_Pwr := 0;
	
	GVL.meter_arr[i].nQuantity_React_Pwr := 4;
	GVL.meter_arr[i].nMBAddr_React_Pwr := 4;
END_FOR

GVL.meter_arr[1].pos := stGRID_POS.pu;
GVL.meter_arr[2].pos := stGRID_POS.poi;

END_FUNCTION_BLOCK

// ---- POUs/Programs/Algorithms/Active power regulation/deltaActivePwr_Frequency_Regulation.TcPOU
FUNCTION deltaActivePwr_Frequency_Regulation : REAL
VAR_INPUT
	p_nd: REAL;
	current_frequency: REAL;
	current_power: REAL;
	//pe_selector: INT;
END_VAR
VAR
	A: stPF_POINT;
	B1: stPF_POINT;
	B2: stPF_POINT;
	DB1: stPF_POINT;
	DB2: stPF_POINT;
	C: stPF_POINT;
	
	p_fn: REAL;
	t: REAL;
	M_LSMO: REAL;
	M_LSMU: REAL;
	pu: REAL;
	max_input: REAL;
	pe: REAL;
	
	B_FSMU: REAL;
	B_FSMO: REAL;
	ActivePwr_Frequency_Regulation: REAL;
END_VAR

//B_FSMU := p_nd * GVL_Freq.K_FSMU; // %
//B_FSMO := p_nd * GVL_Freq.K_FSMO; // %

//p_fn := GVL_Act_Pwr.setpoint;
//M_LSMO := p_fn - B_FSMO;
//pu := p_fn + B_FSMU;

//IF pe_selector = 0 THEN
//	pe := p_nd;
//ELSE 
//	pe := 0;
//END_IF

//M_LSMU := MAX(0, pe - pu);

///// define coordinates ///
//A.frequency := 49.5;
//A.active_power := M_LSMU + p_fn; // = Pfn + Mu

//B1.frequency := 49.8;
//B1.active_power := p_fn + B_FSMU; // = Pfn + Bfsm_u

//DB1.frequency := 49.980;
//DB1.active_power := p_fn; // = Pfn

//DB2.frequency := 50.020;
//DB2.active_power := p_fn; // = Pfn

//B2.frequency := 50.2;
//B2.active_power := p_fn - B_FSMO; // = Pfn - Bfsm_o

//C.frequency := 51.5;
//C.active_power := 0;


////A.frequency := 49.5;
////A.active_power := M_LSMU + p_fn; // = Pfn + Mu

////B1.frequency := -0.2;
////B1.active_power := 0.5; // = Pfn + Bfsm_u

////DB1.frequency := -0.15;
////DB1.active_power := 0; // = Pfn

////DB2.frequency := 0.15;
////DB2.active_power := 0; // = Pfn

////B2.frequency := 0.2;
////B2.active_power := -0.5; // = Pfn - Bfsm_o

////C.frequency := 51.5;
////C.active_power := 0;
////////////////////////////

//IF NOT (current_frequency < DB2.frequency AND current_frequency > DB1.frequency) THEN
	
//	/// SEGMENTO DB2 - B2 ////
//	IF (current_frequency >= DB2.frequency AND current_frequency <= B2.frequency) THEN
//		t := (current_frequency - DB2.frequency) / (B2.frequency - DB2.frequency);
//		ActivePwr_Frequency_Regulation := t*B2.active_power + (1-t)*DB2.active_power;
	
	
//	/// SEGMENTO B2 - C ///
//	ELSIF (current_frequency > B2.frequency AND current_frequency <= C.frequency) THEN
//		t := (current_frequency - B2.frequency) / (C.frequency - B2.frequency);
//		ActivePwr_Frequency_Regulation := t*C.active_power + (1-t)*B2.active_power;
		
	
//	/// Caso limite C ///
//	ELSIF current_frequency > C.frequency THEN
//		ActivePwr_Frequency_Regulation := 0;
		
	
//	/// SEGMENTO B1 - DB1 ///
//	ELSIF (current_frequency >= B1.frequency AND current_frequency <= DB1.frequency) THEN
//		t := (current_frequency - B1.frequency) / (DB1.frequency - B1.frequency);
//		ActivePwr_Frequency_Regulation := t*DB1.active_power + (1-t)*B1.active_power;

	
//	/// SEGMENTO A - B1 ///
//	ELSIF (current_frequency >= A.frequency AND current_frequency <= B1.frequency) THEN
//		t := (current_frequency - A.frequency) / (B1.frequency - A.frequency);
//		ActivePwr_Frequency_Regulation := t*B1.active_power + (1-t)*A.active_power;

	
//	/// Caso limite A ///
//	ELSIF current_frequency < A.frequency THEN
//		/// aggiornare il valore di compensazione  
	
//	END_IF
	
//	deltaActivePwr_Frequency_Regulation := ActivePwr_Frequency_Regulation - GVL_Act_Pwr.setpoint;
	
//ELSE
//	deltaActivePwr_Frequency_Regulation := 0;
//END_IF

//IF deltaActivePwr_Frequency_Regulation > GVL_Freq.out_limiter_max THEN
//	deltaActivePwr_Frequency_Regulation := GVL_Freq.out_limiter_max;
//ELSIF deltaActivePwr_Frequency_Regulation < GVL_Freq.out_limiter_min THEN
//	deltaActivePwr_Frequency_Regulation := GVL_Freq.out_limiter_min;
//END_IF

END_FUNCTION

// ---- POUs/Programs/Algorithms/Cosmo Eco/Calculate_Opt_SOC_Based_On_Conditions.TcPOU
FUNCTION Calculate_Opt_SOC_Based_On_Conditions : REAL
VAR_INPUT
	remaining_battery_capacity: REAL;
	max_diff_per_sample: REAL;
END_VAR
VAR
	optimal_val_for_current_soc: REAL;
	decrease_time: REAL;
	time_to_reach: REAL;
	charge_request: REAL;
END_VAR

optimal_val_for_current_soc := remaining_battery_capacity / 3;
decrease_time := optimal_val_for_current_soc / (max_diff_per_sample * 1200);	// TO DO: parametrizzare
optimal_val_for_current_soc := remaining_battery_capacity / (3+decrease_time + 0.1);

time_to_reach := (GVL.VIRTUAL_METER.active_power_prod - optimal_val_for_current_soc) / (max_diff_per_sample * 1200);
charge_request := ((GVL.VIRTUAL_METER.active_power_prod - optimal_val_for_current_soc) /2 ) * time_to_reach; 

optimal_val_for_current_soc := (remaining_battery_capacity + charge_request)/(3 + decrease_time + 0.1);
optimal_val_for_current_soc := optimal_val_for_current_soc/95*100;

Calculate_Opt_SOC_Based_On_Conditions := optimal_val_for_current_soc;

END_FUNCTION

// ---- POUs/Programs/Algorithms/Cosmo Eco/Calculate_Opt_SOC_No_Decrease.TcPOU
FUNCTION Calculate_Opt_SOC_No_Decrease : REAL
VAR_INPUT
	most_rapid_decrease_h: REAL;
	max_diff_per_sample: REAL;
END_VAR
VAR
	most_rapid_decrease_time: REAL;
	constant_kw_to_support: REAL;
	decrease_avg_kw_to_support: REAL;
	avg_kwh_to_support: REAL;
	decrease_time_found: REAL;
	optimal_soc: REAL;
END_VAR

most_rapid_decrease_time := most_rapid_decrease_h*(GVL.VIRTUAL_METER.active_power_prod / GVL.power_plant.nominal_power);
constant_kw_to_support := GVL.VIRTUAL_POI_METER.active_power_prod;
decrease_avg_kw_to_support := (GVL.VIRTUAL_METER.active_power_prod / 2);

IF GVL.VIRTUAL_POI_METER.active_power_prod > GVL.VIRTUAL_METER.active_power_prod THEN
	
	decrease_avg_kw_to_support := decrease_avg_kw_to_support;

END_IF

avg_kwh_to_support := (constant_kw_to_support * (3 - most_rapid_decrease_time) + decrease_avg_kw_to_support * most_rapid_decrease_time) / 3;
decrease_time_found := (avg_kwh_to_support)/(max_diff_per_sample * 1200);

optimal_soc := avg_kwh_to_support*3+(avg_kwh_to_support*decrease_time_found) / GVL.battery.efficiency;
Calculate_Opt_SOC_No_Decrease := optimal_soc;

END_FUNCTION

// ---- POUs/Programs/Algorithms/Cosmo Eco/Calculate_Set_Point_Normal_Conditions.TcPOU
FUNCTION Calculate_Set_Point_Normal_Conditions : stCMD_SET
VAR_INPUT
END_VAR
VAR
	max_kw_change_3s: REAL;
END_VAR

max_kw_change_3s := (GVL.power_plant.ramp_limit / (60 / GVL.power_plant.sample_time));

IF GVL.battery.soc > GVL.battery.max_tolerable_soc OR (*PowerPlant.ReachingSetPoint*) GVL.battery.soc > GVL.battery.soc_to_remove_sp THEN
	
	IF GVL.VIRTUAL_POI_METER.active_power_prod + max_kw_change_3s < GVL.VIRTUAL_METER.active_power_prod OR (*PowerPlant.ReachingSetPoint AND*) GVL.battery.soc > GVL.battery.soc_to_remove_sp THEN
		
		Calculate_Set_Point_Normal_Conditions := GVL.VIRTUAL_POI_METER.active_power_prod / GVL.power_plant.nominal_power - GVL.power_plant.safety_margin;
		//PowerPlant.ReachingSetPoint := TRUE;
		
	ELSE 
		
		Calculate_Set_Point_Normal_Conditions := -1; 
		RETURN;
		
	END_IF
ELSE
	
	//PowerPlant.ReachingSetPoint := FALSE;
	IF GVL.VIRTUAL_METER.active_power_sp <> 1 THEN
		
		Calculate_Set_Point_Normal_Conditions := 1;
		
	ELSE
 
		Calculate_Set_Point_Normal_Conditions := -2;
	
	END_IF
	
END_IF
RETURN;

END_FUNCTION

// ---- POUs/Programs/Algorithms/Cosmo Eco/No_Decrease.TcPOU
FUNCTION No_Decrease : stCMD_SET
VAR_INPUT
END_VAR
VAR
	remaining_battery_capacity: REAL;
	remaining_limitation_hours: REAL;
	constant_kw_to_support: REAL;
	hours_battery_support: REAL;
	target: REAL;
END_VAR

GVL.power_plant.max_power_increase := GVL.power_plant.ramp_limit/(60/GVL.power_plant.sample_time);
remaining_battery_capacity := (GVL.battery.soc - GVL.battery.min_soc + 0.02) * GVL.battery.capacity; //  TO DO: parametrizzare il margine di sicurezza +0.02 
constant_kw_to_support := (GVL.VIRTUAL_POI_METER.active_power_prod + GVl.power_plant.max_power_increase)/GVL.battery.efficiency;

remaining_limitation_hours := GVL.WISNAM_PPC.timeslot.end - GVL.power_plant.current_time;


IF constant_kw_to_support > 0 THEN
		
	hours_battery_support := (remaining_battery_capacity / constant_kw_to_support);   
		
ELSE
	
	hours_battery_support := 24.0;
		
END_IF
	

	
IF (GVL.VIRTUAL_METER.active_power_prod > GVL.VIRTUAL_POI_METER.active_power_prod) AND (hours_battery_support >= remaining_limitation_hours) THEN		   // If the production is increasing and battery would last enough, we increase the target at POI  
	
	target := GVL.VIRTUAL_POI_METER.active_power_prod + GVL.power_plant.max_power_increase * GVL.battery.soc;
	
	IF target > GVL.power_plant.nominal_power THEN 		
		
		target := GVL.power_plant.nominal_power;			
		
	END_IF
ELSE 
	
	target := GVL.VIRTUAL_POI_METER.active_power_prod; 
END_IF


No_Decrease.command_for_battery := (GVL.VIRTUAL_METER.active_power_prod - target)/(3600/GVL.power_plant.sample_time);
No_Decrease.plant_sp := GVL.VIRTUAL_METER.active_power_prod / GVL.power_plant.nominal_power;


IF GVL.battery.soc > GVL.battery.max_tolerable_soc OR (*(PowerPlant.ReachingSetPoint AND*) GVL.battery.soc > GVl.battery.soc_to_remove_sp THEN		// If battery is too high when entering the timeslot, a setpoint is needed
	
	//PowerPlant.ReachingSetPoint := TRUE;
	No_Decrease.plant_sp := GVL.VIRTUAL_POI_METER.active_power_prod / GVL.power_plant.nominal_power + 0.001;	// TO DO: parametrizzare questo valore

ELSE 
	
	//PowerPlant.ReachingSetPoint := FALSE;
	IF No_Decrease.plant_sp <> 1 THEN
		
		No_Decrease.plant_sp := 1;
	
	ELSE
	
		No_Decrease.plant_sp := -2;
	
	END_IF
END_IF

IF No_Decrease.plant_sp > 1 THEN
	
	No_Decrease.plant_sp := 1;	

END_IF

END_FUNCTION

// ---- POUs/Programs/Algorithms/Cosmo Eco/No_Increase.TcPOU
FUNCTION No_Increase : stCMD_SET
VAR_INPUT
END_VAR
VAR
	target: REAL;
	prod_ratio: REAL;
END_VAR

GVL.power_plant.max_power_increase := GVL.power_plant.ramp_limit/(60/GVL.power_plant.sample_time);
target := GVL.VIRTUAL_POI_METER.active_power_prod;

IF GVL.VIRTUAL_METER.active_power_prod <> 0 THEN
	prod_ratio := GVL.VIRTUAL_POI_METER.active_power_prod / GVL.VIRTUAL_METER.active_power_prod;
END_IF
	
IF GVL.battery.soc < GVL.bess.min_working_soc OR prod_ratio > 2 THEN
	
	target := GVL.VIRTUAL_POI_METER.active_power_prod - GVL.power_plant.max_power_increase * (1 - GVL.battery.soc);
	IF Target < 0 THEN
		Target := 0;
	END_IF

END_IF

No_Increase.command_for_battery := (GVL.VIRTUAL_METER.active_power_prod - target)/(3600 / GVL.power_plant.sample_time);
No_Increase.plant_sp := GVL.VIRTUAL_METER.active_power_prod / GVL.power_plant.nominal_power - GVL.power_plant.safety_margin;

IF GVL.battery.soc > GVL.battery.max_tolerable_soc OR (*PowerPlant.ReachingSetPoint*) GVL.battery.soc > GVL.battery.soc_to_remove_sp THEN          // If the production is increasing and the BESS is already at full charge, we can do nothing but apply a setpoint
	
	// PowerPlant.ReachingSetPoint := TRUE;
	No_Increase.plant_sp := GVL.VIRTUAL_POI_METER.active_power_prod / GVL.power_plant.nominal_power - GVL.power_plant.safety_margin;

ELSE
	// PowerPlant.ReachingSetPoint := FALSE;
	IF No_Increase.plant_sp <> 1 THEN			
	
		No_Increase.plant_sp := 1;
	
	ELSE

		No_Increase.plant_sp := -2; 

	END_IF
END_IF

END_FUNCTION

// ---- POUs/Programs/Algorithms/Cosmo Eco/No_Limit.TcPOU
FUNCTION No_Limit : stCMD_SET
VAR_INPUT
END_VAR
VAR
	max_diff_per_sample: REAL;
	remaining_battery_capacity: REAL;
	constant_kw_to_support: REAL;
	target: REAL;
	hours_battery_support: REAL;
	can_handle_two_hours_prod: BOOL;
	multiplier: REAL;
	max_kw: REAL;
END_VAR

No_Limit.plant_sp := Calculate_Set_Point_Normal_Conditions();
max_diff_per_sample := GVL.power_plant.ramp_limit / (60 / GVL.power_plant.sample_time);
remaining_battery_capacity := (GVL.battery.soc - GVL.battery.min_working_soc) * GVL.battery.capacity;  
constant_kw_to_support := (GVL.power_plant.avg_prod / 3.0) / GVL.battery.efficiency;


IF No_Limit.plant_sp = -1 THEN
    target := GVL.VIRTUAL_POI_METER.active_power_prod + GVL.power_plant.max_power_increase;  
    No_Limit.command_for_battery := (GVL.VIRTUAL_METER.active_power_prod - target) / (3600 / GVL.power_plant.sample_time);
    No_Limit.plant_sp := 1;
    RETURN;
END_IF

IF constant_kw_to_support = 0 THEN
    hours_battery_support := 24; 	
ELSIF constant_kw_to_support > 0 THEN
    hours_battery_support := (remaining_battery_capacity / constant_kw_to_support); 
END_IF


can_handle_two_hours_prod := (hours_battery_support >= 2); 

IF GVL.VIRTUAL_METER.active_power_prod > 0 THEN
    No_Limit.command_for_battery := 0;
    target := GVL.power_plant.avg_prod;

    IF (NOT can_handle_two_hours_prod) AND ((GVL.VIRTUAL_METER.active_power_prod - GVL.VIRTUAL_POI_METER.active_power_prod) > GVL.power_plant.max_power_increase) THEN
        target := GVL.VIRTUAL_POI_METER.active_power_prod;
        
        IF GVL.battery.soc > 0 THEN
            target := target + GVL.power_plant.max_power_increase / 3;
        END_IF
        
        No_Limit.command_for_battery := (GVL.VIRTUAL_METER.active_power_prod - target) / (3600 / GVL.power_plant.sample_time);
        
        IF GVL.battery.soc <= GVL.battery.max_opt_soc AND target >= GVL.VIRTUAL_METER.active_power_prod THEN
            No_Limit.plant_sp := 1;
        END_IF
        RETURN;
    
    ELSE
        IF GVL.battery.soc < GVL.battery.min_opt_soc AND (GVL.VIRTUAL_METER.active_power_prod / GVL.power_plant.nominal_power) > 0.9 THEN
			
            IF (GVL.VIRTUAL_POI_METER.active_power_prod / GVL.power_plant.nominal_power) > 0.80 THEN
                target := GVL.VIRTUAL_POI_METER.active_power_prod - max_diff_per_sample;
            END_IF
			IF GVL.VIRTUAL_POI_METER.active_power_prod / GVL.power_plant.nominal_power < 0.80 THEN
                target := GVL.VIRTUAL_POI_METER.active_power_prod + max_diff_per_sample;
            END_IF
            
            No_Limit.command_for_battery := (GVL.VIRTUAL_METER.active_power_prod - target) / (3600 / GVL.power_plant.sample_time);
            
            IF GVL.battery.soc <= GVL.battery.max_tolerable_soc AND target >= GVL.VIRTUAL_METER.active_power_prod THEN
                No_Limit.plant_sp := 1;
            END_IF
            RETURN;
        
        ELSE
            IF GVL.battery.soc > GVL.battery.max_opt_soc AND can_handle_two_hours_prod THEN
                target := GVL.VIRTUAL_POI_METER.active_power_prod + max_diff_per_sample;
                
                IF target > GVL.power_plant.nominal_power THEN										
                    target := GVL.power_plant.nominal_power;
                END_IF
                
                No_Limit.command_for_battery := (GVL.VIRTUAL_METER.active_power_prod - target) / (3600 / GVL.power_plant.sample_time);
                
                IF GVL.battery.soc <= GVL.battery.max_tolerable_soc AND target >= GVL.VIRTUAL_METER.active_power_prod THEN
                    No_Limit.plant_sp := 1;
                END_IF
                RETURN;			
            END_IF

            IF ABS(GVL.power_plant.avg_prod_diff) > max_diff_per_sample THEN
                IF GVL.power_plant.avg_prod_diff > 0 THEN
                    target := target - (GVL.power_plant.avg_prod_diff - max_diff_per_sample);
                ELSE
                    IF (ABS(GVL.power_plant.avg_prod_diff) / max_diff_per_sample) < 3 OR GVL.battery.soc < 0.4 THEN
                        target := target + ABS(GVL.power_plant.avg_prod_diff) - max_diff_per_sample;
                    ELSE
                        multiplier := SQRT(ABS(GVL.power_plant.avg_prod_diff) / max_diff_per_sample);
                        
                        IF multiplier > 3 THEN			
                            multiplier := 3;
                        END_IF
                        
                        target := target + (multiplier * (ABS(GVL.power_plant.avg_prod_diff) - max_diff_per_sample));
                    END_IF
                END_IF
            END_IF
                    
            IF ABS(GVL.VIRTUAL_POI_METER.active_power_prod - target) > max_diff_per_sample THEN
                IF target > GVL.VIRTUAL_POI_METER.active_power_prod THEN
                    target := GVL.VIRTUAL_POI_METER.active_power_prod + max_diff_per_sample;
                    
                    IF GVL.battery.soc < GVL.battery.min_tolerable_soc AND GVL.battery.soc > 0 THEN	
                        target := GVL.VIRTUAL_POI_METER.active_power_prod - ((max_diff_per_sample) / (1 / GVL.battery.soc));
					END_IF
                    IF GVL.battery.soc = 0 THEN
                        target := GVL.VIRTUAL_POI_METER.active_power_prod - (max_diff_per_sample / 3);
                    END_IF
                    
                ELSE
                    max_kw := GVL.battery.soc * (GVL.battery.capacity / 10);
                    
                    IF GVL.battery.soc > 0.2 AND max_diff_per_sample < max_kw THEN
                        target := GVL.VIRTUAL_POI_METER.active_power_prod - (max_diff_per_sample * (1 - GVL.battery.soc));
                    ELSE
                        target := GVL.VIRTUAL_POI_METER.active_power_prod - max_diff_per_sample;						
                    END_IF
                END_IF			
            END_IF
        END_IF

        IF target < 0 THEN
            target := 0;
        END_IF
        
        No_Limit.command_for_battery := (GVL.VIRTUAL_METER.active_power_prod - target) / (3600 / GVL.power_plant.sample_time);
        
        IF GVL.battery.soc <= GVL.battery.max_tolerable_soc AND target >= GVL.VIRTUAL_METER.active_power_prod THEN
            No_Limit.plant_sp := 1;
        END_IF
        RETURN;	
    END_IF
ELSE
    target := GVL.VIRTUAL_POI_METER.active_power_prod - max_diff_per_sample;

    IF target < 0 THEN 
        target := 0;
    END_IF

    No_Limit.command_for_battery := (GVL.VIRTUAL_METER.active_power_prod - target) / (3600 / GVL.power_plant.sample_time);
    
    IF GVL.battery.soc <= GVL.battery.max_tolerable_soc AND target >= GVL.VIRTUAL_METER.active_power_prod THEN
        No_Limit.plant_sp := 1;
    END_IF
	RETURN;
END_IF

END_FUNCTION

// ---- POUs/Programs/Algorithms/Cosmo Eco/Pre_Lim.TcPOU
FUNCTION Pre_Lim : stCMD_SET
VAR_INPUT
END_VAR
VAR
	max_diff_per_sample: REAL;
	remaining_battery_capacity: REAL;
	remaining_pre_limitation_hours: REAL;
	condition_to_pass: BOOL;
	most_rapid_decrease: REAL;
	constant_kw_to_support: REAL;
	decrease_avg_kw_to_support: REAL;
	avg_kwh_to_support: REAL;
	hours_battery_support: REAL;
	target: REAL;
	decrease_time: REAL;
	prod_ratio: REAL;
	
	opt_soc_value: REAL;
	charge_to_store: REAL;
	time_to_reach_opt_soc: REAL;
	sp_to_send: REAL;
	
	soc_found_for_condition: REAL;
END_VAR

max_diff_per_sample := GVL.power_plant.max_power_increase/(60/GVL.power_plant.sample_time);                // Default calculations
remaining_battery_capacity := (GVL.battery.soc - GVL.battery.min_working_soc)*GVL.battery.capacity;
remaining_pre_limitation_hours := GVL.WISNAM_PPC.timeslot.end - GVL.power_plant.current_time;
condition_to_pass := FALSE;

IF (GVL.WISNAM_PPC.timeslot.next = 'NoDecrease') OR (GVL.WISNAM_PPC.timeslot.next = 'Static') THEN       // Check if the production cannot increase in the upcoming timeslot
	
//	most_rapid_decrease := 1.2*(GVL.VIRTUAL_METER.active_power_prod / GVL.power_plant.nominal_power); //In hours
//	constant_kw_to_support := GVL.VIRTUAL_POI_METER.active_power_prod / GVL.battery.efficiency;		
//	decrease_avg_kw_to_support := GVL.VIRTUAL_METER.active_power_prod / 2;
//	avg_kwh_to_support := (constant_kw_to_support * (3 - most_rapid_decrease) + decrease_avg_kw_to_support * most_rapid_decrease) / 3;  // ??? 3 = SampleTime ??
	
//	IF constant_kw_to_support > 0 THEN
		
//		hours_battery_support := (remaining_battery_capacity / avg_kwh_to_support);
//		//hours_battery_support := (remaining_battery_capacity / constant_kw_to_support);
	
//	ELSE

//		hours_battery_support := 24.0;
	
//	END_IF
	
//	condition_to_pass := (hours_battery_support >= 3);

	soc_found_for_condition := Calculate_Opt_SOC_No_Decrease(most_rapid_decrease_h := 1.2, max_diff_per_sample := max_diff_per_sample);
	condition_to_pass := remaining_battery_capacity > soc_found_for_condition;  
	
	IF (GVL.power_plant.avg_prod_3h > 86000) AND (GVL.power_plant.std_deviation_prod < 10500) AND (remaining_pre_limitation_hours > 0.1) THEN
		
		IF GVL.battery.soc > 0.80 THEN
			
			target := GVL.VIRTUAL_POI_METER.active_power_prod + max_diff_per_sample;
			IF target > GVL.power_plant.nominal_power THEN
				target := GVL.power_plant.nominal_power;
			END_IF
			Pre_Lim.plant_sp := 1;
			IF GVL.battery.soc > GVL.battery.max_tolerable_soc AND target + max_diff_per_sample < GVL.VIRTUAL_METER.active_power_prod THEN
				Pre_Lim.plant_sp := GVL.VIRTUAL_METER.active_power_prod / GVL.power_plant.nominal_power - GVL.power_plant.safety_margin;
			END_IF
			Pre_Lim.plant_sp := (GVL.VIRTUAL_METER.active_power_prod - target)/(3600/GVL.power_plant.sample_time);
			RETURN;
			
		END_IF
		
		IF GVL.battery.soc > 0.7 THEN // 70%??
			
			target := GVL.VIRTUAL_POI_METER.active_power_prod - max_diff_per_sample / 6; // 6?;
			IF target < GVL.power_plant.avg_prod_3h - GVL.power_plant.std_deviation_prod/2 THEN
				target := GVL.power_plant.avg_prod_3h - GVL.power_plant.std_deviation_prod/2;
			END_IF
	 		Pre_Lim.plant_sp := 1;
			IF GVL.battery.soc > GVL.battery.max_tolerable_soc AND (target + max_diff_per_sample) < GVL.VIRTUAL_METER.active_power_prod THEN
				Pre_Lim.plant_sp := GVL.VIRTUAL_METER.active_power_prod / GVL.power_plant.nominal_power - GVL.power_plant.safety_margin;
			END_IF
			Pre_Lim.command_for_battery := (GVL.VIRTUAL_METER.active_power_prod - target)/(3600/GVL.power_plant.sample_time);
			
		END_IF
	
	END_IF
		
ELSE

	constant_kw_to_support := (GVL.VIRTUAL_POI_METER.active_power_prod/2) / GVL.battery.efficiency;
	decrease_time := GVL.VIRTUAL_POI_METER.active_power_prod / (max_diff_per_sample * 3600 / GVL.power_plant.sample_time);
	IF constant_kw_to_support > 0 THEN
		
		hours_battery_support := (remaining_battery_capacity / constant_kw_to_support);
	
	ELSE
		
		hours_battery_support := 24.0;	
	
	END_IF
	
	IF hours_battery_support > decrease_time THEN
		
		condition_to_pass := TRUE;
	
	END_IF
			
END_IF


IF condition_to_pass THEN
	
	IF GVL.battery.soc > GVL.battery.max_tolerable_soc THEN
		Pre_Lim.plant_sp := GVL.VIRTUAL_POI_METER.active_power_prod / GVL.power_plant.nominal_power - 0.005;
	ELSE
		IF GVL_Act_Pwr.total_sp <> 1 THEN
			Pre_Lim.plant_sp := 1;
		ELSE
			Pre_Lim.plant_sp := -2;	
		END_IF
	END_IF
	
	IF (GVL.WISNAM_PPC.timeslot.next = 'NoDecrease') OR (GVL.WISNAM_PPC.timeslot.next = 'Static') THEN
		
		IF GVL.VIRTUAL_POI_METER.active_power_prod <> 0 THEN
			prod_ratio := GVL.VIRTUAL_METER.active_power_prod / GVL.VIRTUAL_POI_METER.active_power_prod;
		END_IF
	
		IF hours_battery_support > 3.2 OR prod_ratio > 1.2 THEN
			
			target := GVL.VIRTUAL_POI_METER.active_power_prod + max_diff_per_sample;
			IF target > GVL.power_plant.nominal_power THEN
				target := GVL.power_plant.nominal_power;
			END_IF
			Pre_Lim.command_for_battery := (GVL.VIRTUAL_METER.active_power_prod - target)/(3600/GVL.power_plant.sample_time);
			IF GVL.battery.soc <= GVL.battery.max_opt_soc AND target >= GVL.VIRTUAL_METER.active_power_prod THEN
				Pre_Lim.plant_sp := 1;
			END_IF
			
			RETURN;
			
		END_IF

	END_IF
	
	Pre_Lim := No_Limit();
	
	RETURN;
	
ELSE 
	
	IF (GVL.WISNAM_PPC.timeslot.next = 'NoDecrease') OR (GVL.WISNAM_PPC.timeslot.next = 'Static') THEN
		
		opt_soc_value := Calculate_Opt_SOC_Based_On_Conditions(remaining_battery_capacity := remaining_battery_capacity, max_diff_per_sample := max_diff_per_sample);
		time_to_reach_opt_soc := (GVL.VIRTUAL_POI_METER.active_power_prod - opt_soc_value) / (max_diff_per_sample * (3600 / GVL.power_plant.sample_time));
		IF remaining_pre_limitation_hours - 0.02 > time_to_reach_opt_soc THEN
			Pre_Lim := No_Limit();
		END_IF
  
	
	END_IF

	target := GVL.power_plant.avg_prod - max_diff_per_sample * (GVL.power_plant.avg_prod_3h / GVL.power_plant.nominal_power);
	
	IF GVL.VIRTUAL_METER.active_power_prod / target > 1.3 OR (GVL.VIRTUAL_POI_METER.active_power_prod < 1000 AND GVL.power_plant.avg_prod_3h > 1000) THEN		// To be removed because too risky?
		target := GVL.VIRTUAL_POI_METER.active_power_prod; 
	END_IF 
	
	IF ABS(GVL.VIRTUAL_POI_METER.active_power_prod - target) > max_diff_per_sample THEN
		
		target := GVL.VIRTUAL_POI_METER.active_power_prod - max_diff_per_sample;
	
	END_IF
	
	sp_to_send := 0;
	
	IF GVL_Act_Pwr.total_sp > (target / GVL.power_plant.nominal_power) + 0.1 THEN
		sp_to_send := target / GVL.power_plant.nominal_power + 0.1;
	END_IF
	

	IF target < 0 THEN
		
		target := 0;
	
	END_IF
	
	Pre_Lim.command_for_battery := (GVL.VIRTUAL_METER.active_power_prod - target) / (3600 / GVL.power_plant.sample_time);
	IF GVL.battery.soc > GVL.battery.max_tolerable_soc THEN
		
		Pre_Lim.plant_sp := GVL.VIRTUAL_POI_METER.active_power_prod / GVL.power_plant.nominal_power - GVL.power_plant.safety_margin;   //  check equation
		
	ELSE
		
		IF GVL_Act_Pwr.total_sp <> 1 THEN
		
			Pre_Lim.plant_sp := 1;

		ELSE
			
			Pre_Lim.plant_sp := -2;		
		
		END_IF
	
	END_IF
	IF GVL.battery.soc <= GVL.battery.max_tolerable_soc AND target >= GVL.VIRTUAL_METER.active_power_prod THEN
		Pre_Lim.plant_sp := 1;
	END_IF
	
END_IF

END_FUNCTION

// ---- POUs/Programs/Algorithms/Cosmo Eco/Static.TcPOU
FUNCTION Static : stCMD_SET
VAR_INPUT
END_VAR
VAR
	target: REAL;
END_VAR

target := GVL.VIRTUAL_POI_METER.active_power_prod;														
Static.command_for_battery := (GVL.VIRTUAL_METER.active_power_prod - Target) / (3600 / GVL.power_plant.sample_time); 
Static.plant_sp := GVL.VIRTUAL_METER.active_power_prod / GVL.power_plant.nominal_power;

IF GVL.battery.soc > GVL.battery.max_tolerable_soc OR (*power_plant.ReachingSetPoint AND *) GVL.battery.soc > GVL.battery.soc_to_remove_sp THEN	// TO DO: capire come implementare la logica del "ReachingSetPoint"
	
	//power_plant.ReachingSetPoint := TRUE;
	Static.plant_sp := (GVL.VIRTUAL_POI_METER.active_power_prod / GVL.power_plant.nominal_power) - GVL.power_plant.safety_margin;    
	
ELSE
	
	//PowerPlant.ReachingSetPoint := FALSE;

	IF Static.plant_sp <> 1 THEN			
		
		Static.plant_sp := 1;
	
	ELSE
	
		Static.plant_sp := -2;	
		
	END_IF 

END_IF

END_FUNCTION

// ---- POUs/Programs/Algorithms/FB_Load_From_DB.TcPOU
FUNCTION_BLOCK FB_Load_From_DB
VAR_INPUT
END_VAR
VAR_OUTPUT
END_VAR
VAR
    bCONNECT: BOOL;
    bEXECUTE: BOOL;
    bREAD : BOOL;
    bDISCONNECT: BOOL;
    
    R_TRIG1: R_TRIG;    
    R_TRIG2: R_TRIG;
    R_TRIG3: R_TRIG;
    R_TRIG4: R_TRIG;
        
    nState: INT;
    nState_Connect: INT;
    nState_Disconnect: INT;
    
    bConn: BOOL;
    bSP: BOOL;    
    bResult: BOOL;
    bData: BOOL;
        
    nDBID: UDINT := 1;
    
    fbSQLDatabase: FB_SQLDatabaseEvt(sNetID:='', tTimeout:=T#10S);
    fbSQLStoredProcedure: FB_SQLStoredProcedureEvt(
                        sNetID:='', tTimeout:=T#10S);
    fbSQLResult: FB_SQLResultEvt(sNetID:='', tTimeout:=T#10S);
    
    arrParameter: ARRAY [0..0] OF ST_SQLSPParameter;
    
    nCustomerID: DINT := 12345;
    
    nRecordStartIndex: UDINT;
    stRecordArr: ARRAY [1..20] OF stRECORD;
    nRecs: UDINT;            
    
    ipResultEvt : Tc3_Eventlogger.I_TcMessage;
    bError : BOOL;
    nEventID: UDINT;
    sEventClass : STRING(255);
    sEventMsg : STRING(255);
END_VAR

//R_TRIG1(CLK:=bCONNECT);
//IF R_TRIG1.Q AND nState = 0 THEN
//    nState := 1;
//END_IF    

//R_TRIG2(CLK:=bEXECUTE);
//IF R_TRIG2.Q AND nState = 0 THEN
//    nState := 2;
//END_IF    

//R_TRIG3(CLK:=bREAD);
//IF R_TRIG3.Q AND nState = 0 THEN
//    nState := 3;
//END_IF

//R_TRIG4(CLK:=bDISCONNECT);
//IF R_TRIG4.Q THEN
//    nState := 4;
//END_IF

//CASE nState OF
//0:(*Idle*)
//    ;
//1: // Connect to database and create stored procedure instance 
//    CASE nState_Connect OF
//        0:
//            IF fbSQLDatabase.Connect(hDBID:= nDBID) THEN
//                ipResultEvt := fbSQLDatabase.ipTcResult;
//                bConn := NOT fbSQLDatabase.bError;
//                IF bConn THEN
//                    nState_Connect := 1;
//                ELSE
//                    nState:=200;
//                END_IF
//            END_IF 
//        1:
//            arrParameter[0].sParameterName := '@Customer_ID';
//            arrParameter[0].eParameterDataType := 
//                            Tc3_Database.E_ColumnType.Integer;
//            arrParameter[0].eParameterType := E_SPParameterType.Input;
//            arrParameter[0].nParameterSize := SIZEOF(nCustomerID);
                        
//            IF fbSQLDatabase.CreateSP('SP_GetAddressByCustomerID',
//                         ADR(arrParameter), SIZEOF(arrParameter),
//                        ADR(fbSQLStoredProcedure)) THEN
//                ipResultEvt:= fbSQLDatabase.ipTcResult;
//                bSP := NOT fbSQLDatabase.bError;
//                nState_Connect:=0;
//                nState := 200;                    
//            END_IF            
//    END_CASE
//2: // Execute stored procedure
//    IF fbSQLStoredProcedure.ExecuteDataReturn(
//                        pParameterStrc:= ADR(nCustomerID),
//                        cbParameterStrc:= SIZEOF(nCustomerID),
//                        pSQLDBResult:= ADR(fbSQLResult)) THEN
//        ipResultEvt:= fbSQLStoredProcedure.ipTcResult;
//        MEMSET(ADR(stRecordArr),0,SIZEOF(stRecordArr));
//        bResult := NOT fbSQLStoredProcedure.bError;
//        nState := 200;            
//    END_IF
//3:    // Read customer positions
//    IF fbSQLResult.Read(nRecordStartIndex, 20, ADR(stRecordArr),
//                    SIZEOF(stRecordArr), TRUE, FALSE) THEN
//        ipResultEvt:= fbSQLResult.ipTcResult;
//        bData := NOT fbSQLStoredProcedure.bError;
//        nRecs := fbSQLResult.nDataCount;
//        nState := 200;                        
//    END_IF
//4:// Disconnect all
//    CASE nState_Disconnect OF
//        0:
//            IF bData THEN
//                IF fbSQLResult.Release() THEN
//                    nState_Disconnect := 1;
//                END_IF
//            ELSE
//                nState_Disconnect := 1;
//            END_IF
//        1:
//            IF bSP THEN
//                IF fbSQLStoredProcedure.Release() THEN
//                    nState_Disconnect := 2;
//                END_IF
//            ELSE
//                nState_Disconnect := 2;
//            END_IF
//        2:
//            IF bConn THEN
//                IF fbSQLDatabase.Disconnect() THEN
//                    nState_Disconnect := 3;
//                END_IF
//            ELSE
//                nState_Disconnect := 3;
//            END_IF
//        3:
//            bData := FALSE;
//            bSP := FALSE;
//            bConn := FALSE;
//            bResult := FALSE;
//            sEventClass := "";
//            sEventMsg := "";
//            nEventID := 0;
//            bError := FALSE;
//            nState_Disconnect := 0;
//            nState := 0;
//    END_CASE
//200:
//    IF ipResultEvt.RequestEventText(1033, sEventMsg, SIZEOF(sEventMsg)) THEN
//        nState := 201;
//    END_IF
//201:
//    IF ipResultEvt.RequestEventClassName(1033, sEventClass, SIZEOF(sEventClass)) THEN

//        nEventID := ipResultEvt.nEventId;

//        bError := (ipResultEvt.eSeverity = TcEventSeverity.Error) OR
//                 (ipResultEvt.eSeverity = TcEventSeverity.Critical);

//        nState:=0;
//    END_IF
//END_CASE

END_FUNCTION_BLOCK

// ---- POUs/Programs/Algorithms/Reactive power regulation/deltaReactivePwr_Voltage_Regulation.TcPOU
FUNCTION deltaReactivePwr_Voltage_Regulation : REAL
VAR_INPUT
	input: REAL;
END_VAR
VAR
	enhancedPoints: ARRAY [1..4, 1..3] OF REAL;
	 i: UINT;
	 x: REAL;
	 y: REAL;
	 g: REAL;
END_VAR

// 8.3.2.1. Regolazione della tensione ad anello aperto – Modalità Q(DV)
enhancedPoints[1][1] := -0.33;
enhancedPoints[1][2] := 0.1;
enhancedPoints[1][3] := -0.3125;

enhancedPoints[2][1] := -0.01;
enhancedPoints[2][2] := 0;
enhancedPoints[2][3] := 0;

enhancedPoints[3][1] := 0.01;
enhancedPoints[3][2] := 0;
enhancedPoints[3][3] := -0.3125;

enhancedPoints[4][1] := 0.33;
enhancedPoints[4][2] := -0.1;
enhancedPoints[4][3] := 0;


x := 0;
y := enhancedPoints[4][2];
g := 0;

IF (input <= enhancedPoints[1][1]) THEN
 	
	x := 0;
	y := enhancedPoints[1][2];
	g := 0;

ELSE 

	FOR i := 4 TO 1 BY -1 DO
		
		IF input < enhancedPoints[i][1] THEN
			CONTINUE;
		END_IF
		
		x := enhancedPoints[i][1];
		y := enhancedPoints[i][2];
		g := enhancedPoints[i][3];
		EXIT;
	
	END_FOR	

END_IF

deltaReactivePwr_Voltage_Regulation := y + g *(input - x);

END_FUNCTION

// ---- POUs/Programs/Engine/Inverter Comm/Apply_Setpoint.TcPOU
FUNCTION_BLOCK Apply_Setpoint
VAR_INPUT
	setpoint: REAL;
	server_port: UINT;
	nUnitID: BYTE;
	nQuantity: WORD;
	nMBAddr: WORD;
	exec_read: BOOL;
END_VAR
VAR_OUTPUT
	bBusy: BOOL;
END_VAR
VAR
	timer_sp: TON;	
	fb_write_holding: FB_MBWriteRegs;
	bError: BOOL;
	nErrId: UDINT;
	ErrId: UDINT;
	aux_union: stCONV_UNION;
	r_trig_exec : R_TRIG; 
END_VAR

aux_union.prod_real := setpoint;

fb_write_holding(
	sIPAddr:= GVL.server_addr, 
	nTCPPort:= server_port, 
	nUnitID:= nUnitID, 
	nQuantity:= nQuantity, 
	nMBAddr:= nMBAddr, 
	cbLength:= SIZEOF(DWORD), 
	pSrcAddr:= ADR(aux_union.prod_w), 
	bExecute:= exec_read, 
	tTimeout:= T#3S, 
	bBusy=> bBusy, 
	bError=> bError, 
	nErrId=> nErrId
);

END_FUNCTION_BLOCK
